  MoveC 1320 to (-42.67, 74.82, -2) mm, rotated rx -180 ry 0 rz 90 deg; joints [75.909, -18.847, 88.976, 0, 19.871, 75.909] to (-41.21, 68.7, -2) mm, rotated rx 180 ry 0 rz 90 deg; joints [75.715, -18.799, 88.77, 0, 20.03, 75.715]
  MoveC 1321 to (-38.99, 66.53, -2) mm, rotated rx 180 ry 0 rz 90 deg; joints [75.66, -18.755, 88.58, 0, 20.175, 75.66] to (-36.48, 64.7, -2) mm, rotated rx -180 ry 0 rz 90 deg; joints [75.62, -18.708, 88.376, 0, 20.331, 75.62]
  MoveL 1322 to (-33.64, 62.89, -2) mm, rotated rx 180 ry 0 rz 90 deg; joints [75.584, -18.654, 88.149, 0, 20.505, 75.584]
  MoveL 1323 to (-13.82, 50.34, -2) mm, rotated rx 180 ry 0 rz 90 deg; joints [75.337, -18.266, 86.548, 0, 21.718, 75.337]
  MoveC 1324 to (-10.3, 48.84, -2) mm, rotated rx -180 ry 0 rz 90 deg; joints [75.318, -18.198, 86.274, 0, 21.924, 75.318] to (-6.48, 48.53, -2) mm, rotated rx 180 ry 0 rz 90 deg; joints [75.34, -18.13, 86.001, 0, 22.129, 75.34]
  MoveL 1325 to (-4.26, 48.7, -2) mm, rotated rx 180 ry 0 rz 90 deg; joints [75.365, -18.091, 85.848, 0, 22.243, 75.365]
  MoveL 1326 to (63.97, 53.62, -2) mm, rotated rx 180 ry 0 rz 90 deg; joints [76.086, -16.793, 80.996, 0, 25.797, 76.086]
  MoveL 1327 to (72, 54.15, -2) mm, rotated rx 180 ry 0 rz 90 deg; joints [76.165, -16.625, 80.404, 0, 26.221, 76.165]
  MoveC 1328 to (76.53, 56.29, -2) mm, rotated rx -180 ry 0 rz 90 deg; joints [76.268, -16.539, 80.104, 0, 26.436, 76.268] to (78.36, 60.94, -2) mm, rotated rx 180 ry 0 rz 90 deg; joints [76.429, -16.524, 80.051, 0, 26.474, 76.429]
  MoveL 1329 to (78.35, 72.49, -2) mm, rotated rx 180 ry 0 rz 90 deg; joints [76.795, -16.584, 80.259, 0, 26.325, 76.795]
  MoveC 1330 to (76.34, 77.27, -2) mm, rotated rx 180 ry 0 rz 90 deg; joints [76.931, -16.651, 80.494, 0, 26.157, 76.931] to (71.55, 79.23, -2) mm, rotated rx 180 ry 0 rz 90 deg; joints [76.958, -16.763, 80.888, 0, 25.875, 76.958]
  MoveC 1331 to (45.96, 79.75, -2) mm, rotated rx 180 ry 0 rz 90 deg; joints [76.784, -17.29, 82.792, 0, 24.498, 76.784] to (20.38, 80.16, -2) mm, rotated rx 180 ry 0 rz 90 deg; joints [76.6, -17.785, 84.654, 0, 23.131, 76.6]
  MoveL 1332 to (20.27, 72.61, -2) mm, rotated rx 180 ry 0 rz 90 deg; joints [76.352, -17.754, 84.532, 0, 23.222, 76.352]
  MoveL 1333 to (20.27, 72.61, 1) mm, rotated rx -180 ry 0 rz 90 deg; joints [76.352, -17.907, 84.632, 0, 23.274, 76.352]
  Establecer velocidad (1000.0 mm/s)
  MoveL 1334 to (20.27, 72.61, 10) mm, rotated rx 180 ry 0 rz 90 deg; joints [76.352, -18.366, 84.932, 0, 23.435, 76.352]
  Establecer velocidad (66.7 mm/s)
  MoveL 1335 to (26.89, 71.36, 10) mm, rotated rx -180 ry 0 rz 90 deg; joints [76.364, -18.234, 84.433, 0, 23.801, 76.364]
  MoveL 1336 to (26.89, 71.36, 1) mm, rotated rx -180 ry 0 rz 90 deg; joints [76.364, -17.776, 84.134, 0, 23.642, 76.364]
  MoveL 1337 to (27.1, 72.86, 0.59) mm, rotated rx -180 ry 0 rz 90 deg; joints [76.415, -17.758, 84.132, 0, 23.626, 76.415]
  MoveL 1338 to (26.94, 74.38, 0.19) mm, rotated rx -180 ry 0 rz 90 deg; joints [76.463, -17.747, 84.156, 0, 23.591, 76.463]
  MoveL 1339 to (26.45, 75.81, -0.22) mm, rotated rx 180 ry 0 rz 90 deg; joints [76.506, -17.743, 84.203, 0, 23.54, 76.506]
  MoveL 1340 to (25.65, 77.11, -0.62) mm, rotated rx -180 ry 0 rz 90 deg; joints [76.542, -17.743, 84.269, 0, 23.474, 76.542]
  MoveL 1341 to (24.58, 78.19, -1.03) mm, rotated rx 180 ry 0 rz 90 deg; joints [76.569, -17.747, 84.351, 0, 23.396, 76.569]
  MoveL 1342 to (23.31, 79.01, -1.44) mm, rotated rx -180 ry 0 rz 90 deg; joints [76.586, -17.754, 84.443, 0, 23.311, 76.586]
  MoveL 1343 to (21.88, 79.53, -1.84) mm, rotated rx 180 ry 0 rz 90 deg; joints [76.591, -17.763, 84.541, 0, 23.222, 76.591]
  MoveL 1344 to (20.37, 79.7, -2.25) mm, rotated rx 180 ry 0 rz 90 deg; joints [76.585, -17.771, 84.638, 0, 23.132, 76.585]
  MoveC 1345 to (-4.74, 80, -2.25) mm, rotated rx 180 ry 0 rz 90 deg; joints [76.396, -18.225, 86.427, 0, 21.799, 76.396] to (-29.85, 80.21, -2.25) mm, rotated rx 180 ry 0 rz 90 deg; joints [76.198, -18.65, 88.179, 0, 20.471, 76.198]
  MoveL 1346 to (-30.8, 80.2, -2.25) mm, rotated rx -180 ry 0 rz 90 deg; joints [76.19, -18.665, 88.244, 0, 20.421, 76.19]
  MoveC 1347 to (-34.29, 79.93, -2.25) mm, rotated rx -180 ry 0 rz 90 deg; joints [76.152, -18.721, 88.48, 0, 20.241, 76.152] to (-37.7, 79.16, -2.25) mm, rotated rx -180 ry 0 rz 90 deg; joints [76.097, -18.772, 88.701, 0, 20.072, 76.097]
  MoveC 1348 to (-42.06, 74.54, -2.25) mm, rotated rx -180 ry 0 rz 90 deg; joints [75.904, -18.823, 88.921, 0, 19.903, 75.904] to (-40.34, 68.41, -2.25) mm, rotated rx 180 ry 0 rz 90 deg; joints [75.712, -18.771, 88.697, 0, 20.074, 75.712]
  MoveC 1349 to (-38.41, 66.69, -2.25) mm, rotated rx -180 ry 0 rz 90 deg; joints [75.671, -18.734, 88.535, 0, 20.199, 75.671] to (-36.32, 65.17, -2.25) mm, rotated rx 180 ry 0 rz 90 deg; joints [75.638, -18.694, 88.365, 0, 20.329, 75.638]
  MoveL 1350 to (-33.64, 63.44, -2.25) mm, rotated rx 180 ry 0 rz 90 deg; joints [75.602, -18.643, 88.15, 0, 20.493, 75.602]
  MoveL 1351 to (-13.47, 50.68, -2.25) mm, rotated rx -180 ry 0 rz 90 deg; joints [75.351, -18.249, 86.522, 0, 21.727, 75.351]
  MoveC 1352 to (-10.21, 49.29, -2.25) mm, rotated rx -180 ry 0 rz 90 deg; joints [75.333, -18.186, 86.268, 0, 21.918, 75.333] to (-6.69, 48.98, -2.25) mm, rotated rx 180 ry 0 rz 90 deg; joints [75.354, -18.123, 86.015, 0, 22.108, 75.354]
  MoveL 1353 to (56.07, 53.54, -2.25) mm, rotated rx 180 ry 0 rz 90 deg; joints [76.021, -16.944, 81.572, 0, 25.372, 76.021]
  MoveL 1354 to (72.01, 54.62, -2.25) mm, rotated rx 180 ry 0 rz 90 deg; joints [76.18, -16.615, 80.404, 0, 26.211, 76.18]
  MoveC 1355 to (76.2, 56.62, -2.25) mm, rotated rx -180 ry 0 rz 90 deg; joints [76.276, -16.536, 80.126, 0, 26.41, 76.276] to (77.91, 60.93, -2.25) mm, rotated rx -180 ry 0 rz 90 deg; joints [76.426, -16.521, 80.076, 0, 26.445, 76.426]
  MoveL 1356 to (77.91, 71.55, -2.25) mm, rotated rx -180 ry 0 rz 90 deg; joints [76.762, -16.576, 80.267, 0, 26.309, 76.762]
  MoveL 1357 to (77.9, 72.49, -2.25) mm, rotated rx 180 ry 0 rz 90 deg; joints [76.792, -16.581, 80.284, 0, 26.297, 76.792]
  MoveC 1358 to (76.02, 76.94, -2.25) mm, rotated rx 180 ry 0 rz 90 deg; joints [76.919, -16.644, 80.504, 0, 26.139, 76.919] to (71.55, 78.78, -2.25) mm, rotated rx -180 ry 0 rz 90 deg; joints [76.944, -16.748, 80.872, 0, 25.876, 76.944]
  MoveC 1359 to (45.96, 79.28, -2.25) mm, rotated rx 180 ry 0 rz 90 deg; joints [76.769, -17.276, 82.776, 0, 24.499, 76.769] to (20.37, 79.7, -2.25) mm, rotated rx 180 ry 0 rz 90 deg; joints [76.585, -17.771, 84.638, 0, 23.132, 76.585]
  MoveL 1360 to (20.26, 72.14, -2.25) mm, rotated rx 180 ry 0 rz 90 deg; joints [76.337, -17.739, 84.516, 0, 23.223, 76.337]
  MoveL 1361 to (20.26, 72.14, 0.75) mm, rotated rx 180 ry 0 rz 90 deg; joints [76.337, -17.892, 84.616, 0, 23.276, 76.337]
  Establecer velocidad (1000.0 mm/s)
  MoveL 1362 to (20.26, 72.14, 10) mm, rotated rx -180 ry 0 rz 90 deg; joints [76.337, -18.364, 84.924, 0, 23.441, 76.337]
  Establecer velocidad (66.7 mm/s)
  MoveL 1363 to (37.42, 27.37, 10) mm, rotated rx -180 ry 0 rz 90 deg; joints [75.031, -17.807, 82.856, 0, 24.951, 75.031]
  MoveL 1364 to (37.42, 27.37, 1) mm, rotated rx 180 ry 0 rz 90 deg; joints [75.031, -17.351, 82.556, 0, 24.795, 75.031]
  MoveL 1365 to (37.57, 28.88, 0.59) mm, rotated rx 180 ry 0 rz 90 deg; joints [75.08, -17.335, 82.561, 0, 24.774, 75.08]
  MoveL 1366 to (37.34, 30.39, 0.19) mm, rotated rx 180 ry 0 rz 90 deg; joints [75.127, -17.327, 82.593, 0, 24.734, 75.127]
  MoveL 1367 to (36.79, 31.8, -0.22) mm, rotated rx -180 ry 0 rz 90 deg; joints [75.167, -17.325, 82.647, 0, 24.678, 75.167]
  MoveL 1368 to (35.94, 33.06, -0.62) mm, rotated rx 180 ry 0 rz 90 deg; joints [75.2, -17.328, 82.72, 0, 24.608, 75.2]
  MoveL 1369 to (34.84, 34.1, -1.03) mm, rotated rx 180 ry 0 rz 90 deg; joints [75.224, -17.335, 82.807, 0, 24.528, 75.224]
  MoveL 1370 to (33.53, 34.87, -1.44) mm, rotated rx 180 ry 0 rz 90 deg; joints [75.238, -17.344, 82.903, 0, 24.441, 75.238]
  MoveL 1371 to (32.08, 35.33, -1.84) mm, rotated rx -180 ry 0 rz 90 deg; joints [75.241, -17.354, 83.003, 0, 24.351, 75.241]
  MoveL 1372 to (30.56, 35.43, -2.25) mm, rotated rx -180 ry 0 rz 90 deg; joints [75.231, -17.364, 83.101, 0, 24.262, 75.231]
  MoveL 1373 to (8.05, 34.82, -2.25) mm, rotated rx 180 ry 0 rz 90 deg; joints [75.018, -17.789, 84.707, 0, 23.081, 75.018]
  MoveL 1374 to (7.11, 34.77, -2.25) mm, rotated rx -180 ry 0 rz 90 deg; joints [75.008, -17.806, 84.774, 0, 23.032, 75.008]
  MoveC 1375 to (3.74, 33.88, -2.25) mm, rotated rx 180 ry 0 rz 90 deg; joints [74.949, -17.863, 84.996, 0, 22.868, 74.949] to (1, 31.75, -2.25) mm, rotated rx 180 ry 0 rz 90 deg; joints [74.856, -17.903, 85.149, 0, 22.753, 74.856]
  MoveC 1376 to (-0.42, 28.07, -2.25) mm, rotated rx 180 ry 0 rz 90 deg; joints [74.723, -17.91, 85.179, 0, 22.731, 74.723] to (0.08, 24.17, -2.25) mm, rotated rx -180 ry 0 rz 90 deg; joints [74.6, -17.882, 85.068, 0, 22.814, 74.6]
  MoveL 1377 to (6.28, 7.11, -2.25) mm, rotated rx 180 ry 0 rz 90 deg; joints [74.103, -17.679, 84.288, 0, 23.391, 74.103]
  MoveC 1378 to (7.37, 5.07, -2.25) mm, rotated rx 180 ry 0 rz 90 deg; joints [74.047, -17.648, 84.169, 0, 23.479, 74.047] to (9, 3.43, -2.25) mm, rotated rx -180 ry 0 rz 90 deg; joints [74.01, -17.609, 84.02, 0, 23.589, 74.01]
  MoveL 1379 to (26.06, -9.85, -2.25) mm, rotated rx -180 ry 0 rz 90 deg; joints [73.742, -17.205, 82.517, 0, 24.688, 73.742]
  MoveL 1380 to (26.62, -10.26, -2.25) mm, rotated rx -180 ry 0 rz 90 deg; joints [73.735, -17.191, 82.467, 0, 24.724, 73.735]
  MoveC 1381 to (31.94, -11.66, -2.25) mm, rotated rx -180 ry 0 rz 90 deg; joints [73.74, -17.077, 82.051, 0, 25.026, 73.74] to (36.8, -9.09, -2.25) mm, rotated rx 180 ry 0 rz 90 deg; joints [73.866, -16.994, 81.751, 0, 25.243, 73.866]
  MoveL 1382 to (37.43, -8.35, -2.25) mm, rotated rx 180 ry 0 rz 90 deg; joints [73.895, -16.986, 81.72, 0, 25.265, 73.895]
  MoveL 1383 to (60.11, 23.22, -2.25) mm, rotated rx 180 ry 0 rz 90 deg; joints [75.091, -16.697, 80.693, 0, 26.004, 75.091]
  MoveC 1384 to (61.33, 25.15, -2.25) mm, rotated rx 180 ry 0 rz 90 deg; joints [75.162, -16.682, 80.64, 0, 26.042, 75.162] to (62.23, 27.25, -2.25) mm, rotated rx 180 ry 0 rz 90 deg; joints [75.236, -16.675, 80.614, 0, 26.061, 75.236]
  MoveC 1385 to (61.82, 32.4, -2.25) mm, rotated rx 180 ry 0 rz 90 deg; joints [75.396, -16.712, 80.745, 0, 25.967, 75.396] to (57.77, 35.62, -2.25) mm, rotated rx 180 ry 0 rz 90 deg; joints [75.464, -16.815, 81.109, 0, 25.706, 75.464]
  MoveC 1386 to (55.91, 35.98, -2.25) mm, rotated rx 180 ry 0 rz 90 deg; joints [75.46, -16.855, 81.254, 0, 25.602, 75.46] to (54.02, 36.06, -2.25) mm, rotated rx -180 ry 0 rz 90 deg; joints [75.447, -16.895, 81.395, 0, 25.5, 75.447]
  MoveL 1387 to (30.56, 35.43, -2.25) mm, rotated rx -180 ry 0 rz 90 deg; joints [75.231, -17.364, 83.101, 0, 24.262, 75.231]
  MoveL 1388 to (30.77, 27.88, -2.25) mm, rotated rx -180 ry 0 rz 90 deg; joints [74.99, -17.32, 82.941, 0, 24.379, 74.99]
  MoveL 1389 to (30.77, 27.88, 0.75) mm, rotated rx 180 ry 0 rz 90 deg; joints [74.99, -17.473, 83.042, 0, 24.431, 74.99]
  Establecer velocidad (1000.0 mm/s)
  MoveL 1390 to (30.77, 27.88, 10) mm, rotated rx 180 ry 0 rz 90 deg; joints [74.99, -17.942, 83.35, 0, 24.592, 74.99]
  Establecer velocidad (66.7 mm/s)
  MoveL 1391 to (70.1, -30.05, 10) mm, rotated rx -180 ry 0 rz 90 deg; joints [73.515, -16.77, 79.233, 0, 27.537, 73.515]
  MoveL 1392 to (70.1, -30.05, 1) mm, rotated rx 180 ry 0 rz 90 deg; joints [73.515, -16.32, 78.931, 0, 27.389, 73.515]
  MoveL 1393 to (71.61, -30.24, 0.59) mm, rotated rx -180 ry 0 rz 90 deg; joints [73.523, -16.265, 78.799, 0, 27.465, 73.523]
  MoveL 1394 to (73.12, -30.06, 0.19) mm, rotated rx 180 ry 0 rz 90 deg; joints [73.542, -16.212, 78.676, 0, 27.536, 73.542]
  MoveL 1395 to (74.55, -29.55, -0.22) mm, rotated rx 180 ry 0 rz 90 deg; joints [73.571, -16.163, 78.565, 0, 27.598, 73.571]
  MoveL 1396 to (75.83, -28.73, -0.62) mm, rotated rx -180 ry 0 rz 90 deg; joints [73.608, -16.119, 78.472, 0, 27.647, 73.608]
  MoveL 1397 to (76.9, -27.65, -1.03) mm, rotated rx -180 ry 0 rz 90 deg; joints [73.651, -16.082, 78.401, 0, 27.681, 73.651]
  MoveL 1398 to (77.7, -26.36, -1.44) mm, rotated rx 180 ry 0 rz 90 deg; joints [73.698, -16.052, 78.355, 0, 27.697, 73.698]
  MoveL 1399 to (78.2, -24.93, -1.84) mm, rotated rx 180 ry 0 rz 90 deg; joints [73.746, -16.03, 78.335, 0, 27.695, 73.746]
  MoveL 1400 to (78.34, -23.41, -2.25) mm, rotated rx 180 ry 0 rz 90 deg; joints [73.794, -16.016, 78.344, 0, 27.672, 73.794]
  MoveL 1401 to (78.34, -5.21, -2.25) mm, rotated rx -180 ry 0 rz 90 deg; joints [74.357, -16.133, 78.739, 0, 27.394, 74.357]
  MoveC 1402 to (78.23, -2.56, -2.25) mm, rotated rx -180 ry 0 rz 90 deg; joints [74.439, -16.152, 78.804, 0, 27.348, 74.439] to (77.84, 0.06, -2.25) mm, rotated rx -180 ry 0 rz 90 deg; joints [74.517, -16.177, 78.888, 0, 27.288, 74.517]
  MoveC 1403 to (74.21, 4.2, -2.25) mm, rotated rx 180 ry 0 rz 90 deg; joints [74.614, -16.282, 79.249, 0, 27.033, 74.614] to (68.7, 4.38, -2.25) mm, rotated rx -180 ry 0 rz 90 deg; joints [74.572, -16.404, 79.668, 0, 26.736, 74.572]
  MoveC 1404 to (66.87, 2.88, -2.25) mm, rotated rx 180 ry 0 rz 90 deg; joints [74.51, -16.434, 79.774, 0, 26.66, 74.51] to (65.31, 1.09, -2.25) mm, rotated rx 180 ry 0 rz 90 deg; joints [74.44, -16.458, 79.854, 0, 26.603, 74.44]
  MoveL 1405 to (64.15, -0.47, -2.25) mm, rotated rx 180 ry 0 rz 90 deg; joints [74.381, -16.473, 79.908, 0, 26.565, 74.381]
  MoveL 1406 to (48.95, -21.32, -2.25) mm, rotated rx 180 ry 0 rz 90 deg; joints [73.592, -16.669, 80.594, 0, 26.075, 73.592]
  MoveL 1407 to (48.51, -21.97, -2.25) mm, rotated rx 180 ry 0 rz 90 deg; joints [73.568, -16.674, 80.613, 0, 26.062, 73.568]
  MoveC 1408 to (47.28, -26.49, -2.25) mm, rotated rx -180 ry 0 rz 90 deg; joints [73.415, -16.672, 80.605, 0, 26.068, 73.415] to (49.04, -30.82, -2.25) mm, rotated rx 180 ry 0 rz 90 deg; joints [73.296, -16.608, 80.378, 0, 26.23, 73.296]
  MoveL 1409 to (49.75, -31.64, -2.25) mm, rotated rx -180 ry 0 rz 90 deg; joints [73.277, -16.588, 80.308, 0, 26.28, 73.277]
  MoveL 1410 to (64.94, -48.8, -2.25) mm, rotated rx 180 ry 0 rz 90 deg; joints [72.888, -16.146, 78.784, 0, 27.362, 72.888]
  MoveL 1411 to (66.07, -50.02, -2.25) mm, rotated rx -180 ry 0 rz 90 deg; joints [72.861, -16.112, 78.67, 0, 27.443, 72.861]
  MoveC 1412 to (67.73, -51.48, -2.25) mm, rotated rx 180 ry 0 rz 90 deg; joints [72.832, -16.066, 78.511, 0, 27.555, 72.832] to (69.65, -52.58, -2.25) mm, rotated rx -180 ry 0 rz 90 deg; joints [72.817, -16.015, 78.34, 0, 27.675, 72.817]
  MoveC 1413 to (75.13, -51.63, -2.25) mm, rotated rx 180 ry 0 rz 90 deg; joints [72.898, -15.898, 77.947, 0, 27.951, 72.898] to (78.06, -46.91, -2.25) mm, rotated rx 180 ry 0 rz 90 deg; joints [73.07, -15.865, 77.834, 0, 28.031, 73.07]
  MoveC 1414 to (78.27, -45.02, -2.25) mm, rotated rx 180 ry 0 rz 90 deg; joints [73.13, -15.873, 77.862, 0, 28.011, 73.13] to (78.34, -43.12, -2.25) mm, rotated rx 180 ry 0 rz 90 deg; joints [73.188, -15.884, 77.9, 0, 27.984, 73.188]
  MoveL 1415 to (78.34, -23.41, -2.25) mm, rotated rx 180 ry 0 rz 90 deg; joints [73.794, -16.016, 78.344, 0, 27.672, 73.794]
  MoveL 1416 to (70.79, -23.41, -2.25) mm, rotated rx -180 ry 0 rz 90 deg; joints [73.726, -16.185, 78.916, 0, 27.269, 73.726]
  MoveL 1417 to (70.79, -23.41, 0.75) mm, rotated rx 180 ry 0 rz 90 deg; joints [73.726, -16.335, 79.018, 0, 27.317, 73.726]
  Establecer velocidad (1000.0 mm/s)
  MoveL 1418 to (70.79, -23.41, 10) mm, rotated rx 180 ry 0 rz 90 deg; joints [73.726, -16.798, 79.328, 0, 27.47, 73.726]
  Establecer velocidad (66.7 mm/s)
  MoveL 1419 to (18.87, -71.64, 10) mm, rotated rx -180 ry 0 rz 90 deg; joints [71.724, -17.584, 82.056, 0, 25.528, 71.724]
  MoveL 1420 to (18.87, -71.64, 1) mm, rotated rx 180 ry 0 rz 90 deg; joints [71.724, -17.129, 81.756, 0, 25.374, 71.724]
  MoveL 1421 to (18.7, -73.15, 0.59) mm, rotated rx -180 ry 0 rz 90 deg; joints [71.675, -17.102, 81.718, 0, 25.384, 71.675]
  MoveL 1422 to (18.9, -74.65, 0.19) mm, rotated rx 180 ry 0 rz 90 deg; joints [71.63, -17.068, 81.654, 0, 25.413, 71.63]
  MoveL 1423 to (19.42, -76.08, -0.22) mm, rotated rx -180 ry 0 rz 90 deg; joints [71.591, -17.027, 81.568, 0, 25.459, 71.591]
  MoveL 1424 to (20.25, -77.35, -0.62) mm, rotated rx 180 ry 0 rz 90 deg; joints [71.56, -16.981, 81.464, 0, 25.517, 71.56]
  MoveL 1425 to (21.34, -78.41, -1.03) mm, rotated rx 180 ry 0 rz 90 deg; joints [71.538, -16.931, 81.345, 0, 25.586, 71.538]
  MoveL 1426 to (22.63, -79.2, -1.44) mm, rotated rx 180 ry 0 rz 90 deg; joints [71.527, -16.879, 81.218, 0, 25.66, 71.527]
  MoveL 1427 to (24.07, -79.69, -1.84) mm, rotated rx -180 ry 0 rz 90 deg; joints [71.527, -16.825, 81.088, 0, 25.737, 71.527]
  MoveL 1428 to (25.59, -79.81, -2.25) mm, rotated rx -180 ry 0 rz 90 deg; joints [71.539, -16.773, 80.961, 0, 25.812, 71.539]
  MoveL 1429 to (46.91, -79.61, -2.25) mm, rotated rx -180 ry 0 rz 90 deg; joints [71.764, -16.325, 79.398, 0, 26.928, 71.764]
  MoveL 1430 to (53.54, -79.52, -2.25) mm, rotated rx 180 ry 0 rz 90 deg; joints [71.833, -16.182, 78.906, 0, 27.276, 71.833]
  MoveC 1431 to (56.29, -79.18, -2.25) mm, rotated rx -180 ry 0 rz 90 deg; joints [71.871, -16.124, 78.709, 0, 27.415, 71.871] to (58.87, -78.18, -2.25) mm, rotated rx 180 ry 0 rz 90 deg; joints [71.928, -16.074, 78.54, 0, 27.534, 71.928]
  MoveC 1432 to (61.62, -73.98, -2.25) mm, rotated rx -180 ry 0 rz 90 deg; joints [72.083, -16.043, 78.435, 0, 27.608, 72.083] to (60.79, -69.03, -2.25) mm, rotated rx -180 ry 0 rz 90 deg; joints [72.227, -16.097, 78.618, 0, 27.479, 72.227]
  MoveC 1433 to (59.74, -67.45, -2.25) mm, rotated rx 180 ry 0 rz 90 deg; joints [72.265, -16.132, 78.735, 0, 27.397, 72.265] to (58.56, -65.96, -2.25) mm, rotated rx -180 ry 0 rz 90 deg; joints [72.299, -16.168, 78.859, 0, 27.309, 72.299]
  MoveL 1434 to (29.78, -32.69, -2.25) mm, rotated rx 180 ry 0 rz 90 deg; joints [73.055, -16.994, 81.751, 0, 25.243, 73.055]
  MoveL 1435 to (28.9, -31.85, -2.25) mm, rotated rx 180 ry 0 rz 90 deg; joints [73.073, -17.017, 81.834, 0, 25.183, 73.073]
  MoveL 1436 to (24.17, -28.06, -2.25) mm, rotated rx 180 ry 0 rz 90 deg; joints [73.147, -17.135, 82.262, 0, 24.873, 73.147]
  MoveL 1437 to (14.55, -20.37, -2.25) mm, rotated rx -180 ry 0 rz 90 deg; joints [73.299, -17.369, 83.123, 0, 24.247, 73.299]
  MoveL 1438 to (13.74, -19.78, -2.25) mm, rotated rx -180 ry 0 rz 90 deg; joints [73.31, -17.388, 83.193, 0, 24.195, 73.31]
  MoveC 1439 to (10.6, -18.25, -2.25) mm, rotated rx -180 ry 0 rz 90 deg; joints [73.329, -17.458, 83.452, 0, 24.006, 73.329] to (7.11, -18.01, -2.25) mm, rotated rx 180 ry 0 rz 90 deg; joints [73.303, -17.525, 83.706, 0, 23.819, 73.303]
  MoveC 1440 to (3.54, -19.84, -2.25) mm, rotated rx 180 ry 0 rz 90 deg; joints [73.21, -17.582, 83.921, 0, 23.662, 73.21] to (1.39, -23.22, -2.25) mm, rotated rx 180 ry 0 rz 90 deg; joints [73.081, -17.604, 84.001, 0, 23.602, 73.081]
  MoveL 1441 to (1.06, -24.17, -2.25) mm, rotated rx 180 ry 0 rz 90 deg; joints [73.047, -17.604, 84.004, 0, 23.601, 73.047]
  MoveL 1442 to (-4.47, -45.01, -2.25) mm, rotated rx 180 ry 0 rz 90 deg; joints [72.326, -17.586, 83.935, 0, 23.651, 72.326]
  MoveL 1443 to (-11.01, -69.65, -2.25) mm, rotated rx -180 ry 0 rz 90 deg; joints [71.474, -17.558, 83.828, 0, 23.73, 71.474]
  MoveL 1444 to (-11.23, -70.6, -2.25) mm, rotated rx -180 ry 0 rz 90 deg; joints [71.441, -17.556, 83.821, 0, 23.735, 71.441]
  MoveC 1445 to (-10.15, -76.46, -2.25) mm, rotated rx 180 ry 0 rz 90 deg; joints [71.267, -17.499, 83.605, 0, 23.893, 71.267] to (-5.21, -79.8, -2.25) mm, rotated rx 180 ry 0 rz 90 deg; joints [71.214, -17.384, 83.176, 0, 24.208, 71.214]
  MoveC 1446 to (-3.8, -80.03, -2.25) mm, rotated rx -180 ry 0 rz 90 deg; joints [71.223, -17.355, 83.07, 0, 24.285, 71.223] to (-2.37, -80.08, -2.25) mm, rotated rx -180 ry 0 rz 90 deg; joints [71.236, -17.327, 82.967, 0, 24.36, 71.236]
  MoveL 1447 to (25.59, -79.81, -2.25) mm, rotated rx -180 ry 0 rz 90 deg; joints [71.539, -16.773, 80.961, 0, 25.812, 71.539]
  MoveL 1448 to (25.51, -72.27, -2.25) mm, rotated rx 180 ry 0 rz 90 deg; joints [71.773, -16.826, 81.149, 0, 25.677, 71.773]
  MoveL 1449 to (25.51, -72.27, 0.75) mm, rotated rx -180 ry 0 rz 90 deg; joints [71.773, -16.977, 81.25, 0, 25.727, 71.773]
  Establecer velocidad (1000.0 mm/s)
  MoveL 1450 to (25.51, -72.27, 10) mm, rotated rx -180 ry 0 rz 90 deg; joints [71.773, -17.444, 81.559, 0, 25.885, 71.773]
  Establecer velocidad (66.7 mm/s)
  MoveL 1451 to (-60.11, -71.82, 10) mm, rotated rx 180 ry 0 rz 90 deg; joints [70.867, -19.042, 87.581, 0, 21.461, 70.867]
  MoveL 1452 to (-60.11, -71.82, 1) mm, rotated rx 180 ry 0 rz 90 deg; joints [70.867, -18.577, 87.282, 0, 21.295, 70.867]
  MoveL 1453 to (-60.28, -73.32, 0.59) mm, rotated rx 180 ry 0 rz 90 deg; joints [70.816, -18.55, 87.245, 0, 21.305, 70.816]
  MoveL 1454 to (-60.09, -74.83, 0.19) mm, rotated rx 180 ry 0 rz 90 deg; joints [70.769, -18.517, 87.182, 0, 21.335, 70.769]
  MoveL 1455 to (-59.57, -76.26, -0.22) mm, rotated rx 180 ry 0 rz 90 deg; joints [70.729, -18.479, 87.099, 0, 21.38, 70.729]
  MoveL 1456 to (-58.74, -77.54, -0.62) mm, rotated rx 180 ry 0 rz 90 deg; joints [70.697, -18.437, 87, 0, 21.438, 70.697]
  MoveL 1457 to (-57.65, -78.6, -1.03) mm, rotated rx -180 ry 0 rz 90 deg; joints [70.675, -18.392, 86.887, 0, 21.505, 70.675]
  MoveL 1458 to (-56.36, -79.39, -1.44) mm, rotated rx 180 ry 0 rz 90 deg; joints [70.664, -18.345, 86.766, 0, 21.579, 70.664]
  MoveL 1459 to (-54.92, -79.88, -1.84) mm, rotated rx 180 ry 0 rz 90 deg; joints [70.664, -18.297, 86.643, 0, 21.654, 70.664]
  MoveL 1460 to (-53.41, -80.01, -2.25) mm, rotated rx 180 ry 0 rz 90 deg; joints [70.677, -18.249, 86.523, 0, 21.726, 70.677]
  MoveL 1461 to (-35.27, -79.87, -2.25) mm, rotated rx -180 ry 0 rz 90 deg; joints [70.885, -17.936, 85.28, 0, 22.656, 70.885]
  MoveC 1462 to (-29.73, -77.98, -2.25) mm, rotated rx -180 ry 0 rz 90 deg; joints [71.006, -17.849, 84.941, 0, 22.908, 71.006] to (-26.4, -73.16, -2.25) mm, rotated rx -180 ry 0 rz 90 deg; joints [71.196, -17.819, 84.824, 0, 22.994, 71.196]
  MoveL 1463 to (-26.21, -72.49, -2.25) mm, rotated rx 180 ry 0 rz 90 deg; joints [71.22, -17.82, 84.827, 0, 22.993, 71.22]
  MoveL 1464 to (-13.74, -24.57, -2.25) mm, rotated rx -180 ry 0 rz 90 deg; joints [72.889, -17.875, 85.041, 0, 22.834, 72.889]
  MoveL 1465 to (-13.64, -24.17, -2.25) mm, rotated rx 180 ry 0 rz 90 deg; joints [72.903, -17.875, 85.042, 0, 22.833, 72.903]
  MoveC 1466 to (-13.44, -19.72, -2.25) mm, rotated rx 180 ry 0 rz 90 deg; joints [73.048, -17.896, 85.123, 0, 22.773, 73.048] to (-15.2, -15.64, -2.25) mm, rotated rx 180 ry 0 rz 90 deg; joints [73.163, -17.95, 85.334, 0, 22.616, 73.163]
  MoveC 1467 to (-19.03, -13.05, -2.25) mm, rotated rx 180 ry 0 rz 90 deg; joints [73.21, -18.032, 85.657, 0, 22.375, 73.21] to (-23.65, -12.75, -2.25) mm, rotated rx -180 ry 0 rz 90 deg; joints [73.174, -18.115, 85.985, 0, 22.13, 73.174]
  MoveL 1468 to (-26.06, -13.23, -2.25) mm, rotated rx 180 ry 0 rz 90 deg; joints [73.134, -18.155, 86.142, 0, 22.012, 73.134]
  MoveL 1469 to (-73.46, -23.33, -2.25) mm, rotated rx 180 ry 0 rz 90 deg; joints [72.316, -18.878, 89.16, 0, 19.718, 72.316]
  MoveC 1470 to (-78.73, -26.56, -2.25) mm, rotated rx 180 ry 0 rz 90 deg; joints [72.152, -18.943, 89.443, 0, 19.5, 72.152] to (-80.79, -32.38, -2.25) mm, rotated rx 180 ry 0 rz 90 deg; joints [71.935, -18.945, 89.455, 0, 19.491, 71.935]
  MoveL 1471 to (-80.79, -70.98, -2.25) mm, rotated rx -180 ry 0 rz 90 deg; joints [70.658, -18.745, 88.583, 0, 20.162, 70.658]
  MoveC 1472 to (-78.08, -77.49, -2.25) mm, rotated rx -180 ry 0 rz 90 deg; joints [70.476, -18.667, 88.249, 0, 20.418, 70.476] to (-71.54, -80.15, -2.25) mm, rotated rx 180 ry 0 rz 90 deg; joints [70.465, -18.548, 87.748, 0, 20.8, 70.465]
  MoveL 1473 to (-53.41, -80.01, -2.25) mm, rotated rx 180 ry 0 rz 90 deg; joints [70.677, -18.249, 86.523, 0, 21.726, 70.677]
  MoveL 1474 to (-53.47, -72.46, -2.25) mm, rotated rx 180 ry 0 rz 90 deg; joints [70.92, -18.295, 86.706, 0, 21.588, 70.92]
  MoveL 1475 to (-53.47, -72.46, 0.75) mm, rotated rx 180 ry 0 rz 90 deg; joints [70.92, -18.449, 86.807, 0, 21.642, 70.92]
  Establecer velocidad (1000.0 mm/s)
  MoveL 1476 to (-53.47, -72.46, 10) mm, rotated rx 180 ry 0 rz 90 deg; joints [70.92, -18.926, 87.114, 0, 21.812, 70.92]
  Establecer velocidad (66.7 mm/s)
  MoveL 1477 to (-72.55, 36.29, 10) mm, rotated rx 180 ry 0 rz 90 deg; joints [74.332, -19.775, 90.703, 0, 19.073, 74.332]
  MoveL 1478 to (-72.55, 36.29, 1) mm, rotated rx 180 ry 0 rz 90 deg; joints [74.332, -19.304, 90.403, 0, 18.9, 74.332]
  MoveL 1479 to (-74.05, 36.47, 0.59) mm, rotated rx -180 ry 0 rz 90 deg; joints [74.324, -19.305, 90.494, 0, 18.811, 74.324]
  MoveL 1480 to (-75.56, 36.29, 0.19) mm, rotated rx 180 ry 0 rz 90 deg; joints [74.303, -19.305, 90.578, 0, 18.728, 74.303]
  MoveL 1481 to (-76.99, 35.78, -0.22) mm, rotated rx 180 ry 0 rz 90 deg; joints [74.272, -19.303, 90.65, 0, 18.653, 74.272]
  MoveL 1482 to (-78.28, 34.96, -0.62) mm, rotated rx -180 ry 0 rz 90 deg; joints [74.232, -19.297, 90.706, 0, 18.59, 74.232]
  MoveL 1483 to (-79.34, 33.88, -1.03) mm, rotated rx 180 ry 0 rz 90 deg; joints [74.185, -19.286, 90.743, 0, 18.543, 74.185]
  MoveL 1484 to (-80.15, 32.59, -1.44) mm, rotated rx -180 ry 0 rz 90 deg; joints [74.133, -19.271, 90.759, 0, 18.512, 74.133]
  MoveL 1485 to (-80.65, 31.16, -1.84) mm, rotated rx -180 ry 0 rz 90 deg; joints [74.079, -19.251, 90.751, 0, 18.5, 74.079]
  MoveL 1486 to (-80.79, 29.64, -2.25) mm, rotated rx -180 ry 0 rz 90 deg; joints [74.026, -19.226, 90.718, 0, 18.508, 74.026]
  MoveL 1487 to (-80.78, 0.47, -2.25) mm, rotated rx -180 ry 0 rz 90 deg; joints [73.037, -19.1, 90.144, 0, 18.955, 73.037]
  MoveC 1488 to (-77.75, -6.36, -2.25) mm, rotated rx -180 ry 0 rz 90 deg; joints [72.838, -19.024, 89.803, 0, 19.221, 72.838] to (-70.6, -8.55, -2.25) mm, rotated rx -180 ry 0 rz 90 deg; joints [72.839, -18.905, 89.279, 0, 19.626, 72.839]
  MoveL 1489 to (-69.65, -8.43, -2.25) mm, rotated rx -180 ry 0 rz 90 deg; joints [72.853, -18.892, 89.218, 0, 19.673, 72.853]
  MoveL 1490 to (-63.02, -6.92, -2.25) mm, rotated rx 180 ry 0 rz 90 deg; joints [72.971, -18.796, 88.803, 0, 19.993, 72.971]
  MoveL 1491 to (-19.43, 3.11, -2.25) mm, rotated rx 180 ry 0 rz 90 deg; joints [73.733, -18.124, 86.019, 0, 22.105, 73.733]
  MoveC 1492 to (-13.57, 7.44, -2.25) mm, rotated rx 180 ry 0 rz 90 deg; joints [73.929, -18.042, 85.697, 0, 22.345, 73.929] to (-12.82, 14.69, -2.25) mm, rotated rx 180 ry 0 rz 90 deg; joints [74.173, -18.066, 85.79, 0, 22.276, 74.173]
  MoveL 1493 to (-13.12, 15.64, -2.25) mm, rotated rx 180 ry 0 rz 90 deg; joints [74.201, -18.076, 85.83, 0, 22.246, 74.201]
  MoveL 1494 to (-19.79, 34.25, -2.25) mm, rotated rx 180 ry 0 rz 90 deg; joints [74.752, -18.282, 86.657, 0, 21.626, 74.752]
  MoveC 1495 to (-21.29, 36.95, -2.25) mm, rotated rx 180 ry 0 rz 90 deg; joints [74.828, -18.321, 86.812, 0, 21.509, 74.828] to (-23.58, 39.01, -2.25) mm, rotated rx -180 ry 0 rz 90 deg; joints [74.876, -18.369, 87.01, 0, 21.359, 74.876]
  MoveL 1496 to (-65.41, 65.86, -2.25) mm, rotated rx -180 ry 0 rz 90 deg; joints [75.406, -19.146, 90.352, 0, 18.794, 75.406]
  MoveL 1497 to (-66.15, 66.33, -2.25) mm, rotated rx -180 ry 0 rz 90 deg; joints [75.416, -19.158, 90.41, 0, 18.749, 75.416]
  MoveC 1498 to (-69.29, 67.73, -2.25) mm, rotated rx 180 ry 0 rz 90 deg; joints [75.436, -19.21, 90.645, 0, 18.565, 75.436] to (-72.7, 68.19, -2.25) mm, rotated rx 180 ry 0 rz 90 deg; joints [75.421, -19.261, 90.881, 0, 18.38, 75.421]
  MoveC 1499 to (-76.86, 66.93, -2.25) mm, rotated rx -180 ry 0 rz 90 deg; joints [75.34, -19.316, 91.136, 0, 18.179, 75.34] to (-79.72, 63.66, -2.25) mm, rotated rx -180 ry 0 rz 90 deg; joints [75.202, -19.344, 91.269, 0, 18.075, 75.202]
  MoveC 1500 to (-80.52, 61.3, -2.25) mm, rotated rx -180 ry 0 rz 90 deg; joints [75.113, -19.347, 91.281, 0, 18.066, 75.113] to (-80.79, 58.82, -2.25) mm, rotated rx 180 ry 0 rz 90 deg; joints [75.025, -19.341, 91.255, 0, 18.086, 75.025]
  MoveL 1501 to (-80.79, 29.64, -2.25) mm, rotated rx -180 ry 0 rz 90 deg; joints [74.026, -19.226, 90.718, 0, 18.508, 74.026]
  MoveL 1502 to (-73.24, 29.65, -2.25) mm, rotated rx -180 ry 0 rz 90 deg; joints [74.1, -19.116, 90.215, 0, 18.901, 74.1]
  MoveL 1503 to (-73.24, 29.65, 0.75) mm, rotated rx -180 ry 0 rz 90 deg; joints [74.1, -19.273, 90.316, 0, 18.957, 74.1]
  Establecer velocidad (1000.0 mm/s)
  MoveL 1504 to (-73.24, 29.65, 10) mm, rotated rx 180 ry 0 rz 90 deg; joints [74.1, -19.758, 90.623, 0, 19.134, 74.1]
  Establecer velocidad (66.7 mm/s)
  MoveL 1505 to (-72.12, 36.29, 10) mm, rotated rx -180 ry 0 rz 90 deg; joints [74.336, -19.769, 90.674, 0, 19.095, 74.336]
  MoveL 1506 to (-72.12, 36.29, 0.75) mm, rotated rx -180 ry 0 rz 90 deg; joints [74.336, -19.284, 90.366, 0, 18.918, 74.336]
  MoveL 1507 to (-73.62, 36.47, 0.34) mm, rotated rx 180 ry 0 rz 90 deg; joints [74.328, -19.286, 90.457, 0, 18.829, 74.328]
  MoveL 1508 to (-75.13, 36.29, -0.06) mm, rotated rx 180 ry 0 rz 90 deg; joints [74.307, -19.286, 90.541, 0, 18.745, 74.307]
  MoveL 1509 to (-76.57, 35.78, -0.47) mm, rotated rx -180 ry 0 rz 90 deg; joints [74.276, -19.283, 90.613, 0, 18.67, 74.276]
  MoveL 1510 to (-77.85, 34.96, -0.87) mm, rotated rx -180 ry 0 rz 90 deg; joints [74.236, -19.277, 90.669, 0, 18.608, 74.236]
  MoveL 1511 to (-78.92, 33.88, -1.28) mm, rotated rx 180 ry 0 rz 90 deg; joints [74.189, -19.267, 90.706, 0, 18.561, 74.189]
  MoveL 1512 to (-79.72, 32.59, -1.69) mm, rotated rx 180 ry 0 rz 90 deg; joints [74.137, -19.252, 90.722, 0, 18.53, 74.137]
  MoveL 1513 to (-80.22, 31.16, -2.09) mm, rotated rx 180 ry 0 rz 90 deg; joints [74.083, -19.232, 90.714, 0, 18.518, 74.083]
  MoveL 1514 to (-80.36, 29.64, -2.5) mm, rotated rx 180 ry 0 rz 90 deg; joints [74.03, -19.206, 90.681, 0, 18.525, 74.03]
  MoveL 1515 to (-80.36, 0.47, -2.5) mm, rotated rx 180 ry 0 rz 90 deg; joints [73.041, -19.081, 90.108, 0, 18.973, 73.041]
  MoveC 1516 to (-78.13, -5.38, -2.5) mm, rotated rx 180 ry 0 rz 90 deg; joints [72.867, -19.021, 89.84, 0, 19.181, 72.867] to (-72.49, -8.11, -2.5) mm, rotated rx 180 ry 0 rz 90 deg; joints [72.834, -18.923, 89.407, 0, 19.516, 72.834]
  MoveL 1517 to (-72.02, -8.13, -2.5) mm, rotated rx -180 ry 0 rz 90 deg; joints [72.838, -18.916, 89.375, 0, 19.541, 72.838]
  MoveC 1518 to (-70.49, -8.09, -2.5) mm, rotated rx 180 ry 0 rz 90 deg; joints [72.856, -18.893, 89.273, 0, 19.62, 72.856] to (-68.97, -7.84, -2.5) mm, rotated rx -180 ry 0 rz 90 deg; joints [72.879, -18.871, 89.176, 0, 19.695, 72.879]
  MoveL 1519 to (-19.43, 3.56, -2.5) mm, rotated rx 180 ry 0 rz 90 deg; joints [73.747, -18.113, 86.02, 0, 22.093, 73.747]
  MoveC 1520 to (-13.88, 7.76, -2.5) mm, rotated rx -180 ry 0 rz 90 deg; joints [73.937, -18.037, 85.717, 0, 22.32, 73.937] to (-13.26, 14.69, -2.5) mm, rotated rx -180 ry 0 rz 90 deg; joints [74.169, -18.061, 85.812, 0, 22.249, 74.169]
  MoveL 1521 to (-13.58, 15.64, -2.5) mm, rotated rx 180 ry 0 rz 90 deg; joints [74.197, -18.071, 85.854, 0, 22.218, 74.197]
  MoveL 1522 to (-20.17, 34.04, -2.5) mm, rotated rx 180 ry 0 rz 90 deg; joints [74.742, -18.275, 86.67, 0, 21.605, 74.742]
  MoveC 1523 to (-21.63, 36.68, -2.5) mm, rotated rx 180 ry 0 rz 90 deg; joints [74.816, -18.312, 86.822, 0, 21.49, 74.816] to (-23.87, 38.7, -2.5) mm, rotated rx 180 ry 0 rz 90 deg; joints [74.863, -18.36, 87.016, 0, 21.344, 74.863]
  MoveL 1524 to (-66.23, 65.86, -2.5) mm, rotated rx -180 ry 0 rz 90 deg; joints [75.399, -19.145, 90.398, 0, 18.746, 75.399]
  MoveC 1525 to (-69.05, 67.21, -2.5) mm, rotated rx 180 ry 0 rz 90 deg; joints [75.42, -19.191, 90.611, 0, 18.58, 75.42] to (-72.13, 67.77, -2.5) mm, rotated rx 180 ry 0 rz 90 deg; joints [75.412, -19.238, 90.827, 0, 18.411, 75.412]
  MoveC 1526 to (-76.69, 66.52, -2.5) mm, rotated rx -180 ry 0 rz 90 deg; joints [75.328, -19.299, 91.109, 0, 18.189, 75.328] to (-79.62, 62.81, -2.5) mm, rotated rx -180 ry 0 rz 90 deg; joints [75.173, -19.326, 91.24, 0, 18.087, 75.173]
  MoveC 1527 to (-80.18, 60.77, -2.5) mm, rotated rx -180 ry 0 rz 90 deg; joints [75.098, -19.327, 91.24, 0, 18.086, 75.098] to (-80.36, 58.67, -2.5) mm, rotated rx 180 ry 0 rz 90 deg; joints [75.024, -19.321, 91.215, 0, 18.106, 75.024]
  MoveL 1528 to (-80.36, 29.64, -2.5) mm, rotated rx 180 ry 0 rz 90 deg; joints [74.03, -19.206, 90.681, 0, 18.525, 74.03]
  MoveL 1529 to (-72.81, 29.65, -2.5) mm, rotated rx 180 ry 0 rz 90 deg; joints [74.104, -19.096, 90.178, 0, 18.918, 74.104]
  MoveL 1530 to (-72.81, 29.65, 0.5) mm, rotated rx -180 ry 0 rz 90 deg; joints [74.104, -19.253, 90.279, 0, 18.975, 74.104]
  Establecer velocidad (1000.0 mm/s)
  MoveL 1531 to (-72.81, 29.65, 10) mm, rotated rx -180 ry 0 rz 90 deg; joints [74.104, -19.751, 90.595, 0, 19.157, 74.104]
  Establecer velocidad (66.7 mm/s)
  MoveL 1532 to (-72.12, -45.33, 10) mm, rotated rx 180 ry 0 rz 90 deg; joints [71.6, -19.384, 88.998, 0, 20.386, 71.6]
  MoveL 1533 to (-72.12, -45.33, 0.75) mm, rotated rx 180 ry 0 rz 90 deg; joints [71.6, -18.903, 88.691, 0, 20.212, 71.6]
  MoveL 1534 to (-73.63, -45.15, 0.34) mm, rotated rx 180 ry 0 rz 90 deg; joints [71.59, -18.906, 88.782, 0, 20.124, 71.59]
  MoveL 1535 to (-75.14, -45.33, -0.06) mm, rotated rx 180 ry 0 rz 90 deg; joints [71.567, -18.907, 88.865, 0, 20.042, 71.567]
  MoveL 1536 to (-76.57, -45.84, -0.47) mm, rotated rx 180 ry 0 rz 90 deg; joints [71.535, -18.906, 88.936, 0, 19.97, 71.535]
  MoveL 1537 to (-77.85, -46.66, -0.87) mm, rotated rx 180 ry 0 rz 90 deg; joints [71.493, -18.9, 88.99, 0, 19.91, 71.493]
  MoveL 1538 to (-78.92, -47.74, -1.28) mm, rotated rx 180 ry 0 rz 90 deg; joints [71.446, -18.89, 89.024, 0, 19.866, 71.446]
  MoveL 1539 to (-79.72, -49.02, -1.69) mm, rotated rx 180 ry 0 rz 90 deg; joints [71.394, -18.875, 89.035, 0, 19.84, 71.394]
  MoveL 1540 to (-80.22, -50.46, -2.09) mm, rotated rx -180 ry 0 rz 90 deg; joints [71.341, -18.854, 89.022, 0, 19.831, 71.341]
  MoveL 1541 to (-80.36, -51.97, -2.5) mm, rotated rx -180 ry 0 rz 90 deg; joints [71.29, -18.827, 88.984, 0, 19.843, 71.29]
  MoveL 1542 to (-80.36, -70.6, -2.5) mm, rotated rx 180 ry 0 rz 90 deg; joints [70.676, -18.727, 88.555, 0, 20.172, 70.676]
  MoveL 1543 to (-80.32, -71.55, -2.5) mm, rotated rx 180 ry 0 rz 90 deg; joints [70.645, -18.722, 88.531, 0, 20.191, 70.645]
  MoveC 1544 to (-77.55, -77.37, -2.5) mm, rotated rx -180 ry 0 rz 90 deg; joints [70.486, -18.646, 88.208, 0, 20.438, 70.486] to (-71.55, -79.73, -2.5) mm, rotated rx 180 ry 0 rz 90 deg; joints [70.479, -18.537, 87.749, 0, 20.788, 70.479]
  MoveL 1545 to (-70.6, -79.73, -2.5) mm, rotated rx -180 ry 0 rz 90 deg; joints [70.49, -18.522, 87.686, 0, 20.836, 70.49]
  MoveL 1546 to (-36.48, -79.45, -2.5) mm, rotated rx 180 ry 0 rz 90 deg; joints [70.885, -17.948, 85.366, 0, 22.582, 70.885]
  MoveL 1547 to (-35.25, -79.44, -2.5) mm, rotated rx -180 ry 0 rz 90 deg; joints [70.899, -17.926, 85.281, 0, 22.645, 70.899]
  MoveC 1548 to (-29.85, -77.53, -2.5) mm, rotated rx -180 ry 0 rz 90 deg; joints [71.019, -17.841, 84.952, 0, 22.889, 71.019] to (-26.71, -72.74, -2.5) mm, rotated rx 180 ry 0 rz 90 deg; joints [71.207, -17.814, 84.848, 0, 22.967, 71.207]
  MoveL 1549 to (-14.07, -24.17, -2.5) mm, rotated rx -180 ry 0 rz 90 deg; joints [72.898, -17.87, 85.064, 0, 22.806, 72.898]
  MoveC 1550 to (-13.81, -20.28, -2.5) mm, rotated rx -180 ry 0 rz 90 deg; joints [73.027, -17.887, 85.129, 0, 22.758, 73.027] to (-15.04, -16.58, -2.5) mm, rotated rx -180 ry 0 rz 90 deg; joints [73.134, -17.929, 85.295, 0, 22.635, 73.134]
  MoveC 1551 to (-18.62, -13.65, -2.5) mm, rotated rx -180 ry 0 rz 90 deg; joints [73.194, -18.009, 85.607, 0, 22.402, 73.194] to (-23.22, -13.12, -2.5) mm, rotated rx 180 ry 0 rz 90 deg; joints [73.166, -18.093, 85.939, 0, 22.154, 73.166]
  MoveL 1552 to (-24.17, -13.28, -2.5) mm, rotated rx 180 ry 0 rz 90 deg; joints [73.152, -18.108, 86.001, 0, 22.107, 73.152]
  MoveL 1553 to (-73.35, -23.74, -2.5) mm, rotated rx -180 ry 0 rz 90 deg; joints [72.303, -18.862, 89.136, 0, 19.726, 72.303]
  MoveC 1554 to (-78.39, -26.82, -2.5) mm, rotated rx 180 ry 0 rz 90 deg; joints [72.146, -18.923, 89.406, 0, 19.517, 72.146] to (-80.36, -32.39, -2.5) mm, rotated rx -180 ry 0 rz 90 deg; joints [71.939, -18.926, 89.417, 0, 19.508, 71.939]
  MoveL 1555 to (-80.36, -51.97, -2.5) mm, rotated rx -180 ry 0 rz 90 deg; joints [71.29, -18.827, 88.984, 0, 19.843, 71.29]
  MoveL 1556 to (-72.81, -51.97, -2.5) mm, rotated rx -180 ry 0 rz 90 deg; joints [71.374, -18.71, 88.479, 0, 20.231, 71.374]
  MoveL 1557 to (-72.81, -51.97, 0.5) mm, rotated rx 180 ry 0 rz 90 deg; joints [71.374, -18.865, 88.579, 0, 20.286, 71.374]
  Establecer velocidad (1000.0 mm/s)
  MoveL 1558 to (-72.81, -51.97, 10) mm, rotated rx -180 ry 0 rz 90 deg; joints [71.374, -19.359, 88.895, 0, 20.464, 71.374]
  Establecer velocidad (66.7 mm/s)
  MoveL 1559 to (18.62, -71.21, 10) mm, rotated rx -180 ry 0 rz 90 deg; joints [71.735, -17.592, 82.084, 0, 25.508, 71.735]
  MoveL 1560 to (18.62, -71.21, 0.75) mm, rotated rx 180 ry 0 rz 90 deg; joints [71.735, -17.125, 81.776, 0, 25.349, 71.735]
  MoveL 1561 to (18.45, -72.72, 0.34) mm, rotated rx 180 ry 0 rz 90 deg; joints [71.686, -17.097, 81.738, 0, 25.359, 71.686]
  MoveL 1562 to (18.65, -74.23, -0.06) mm, rotated rx -180 ry 0 rz 90 deg; joints [71.641, -17.063, 81.674, 0, 25.389, 71.641]
  MoveL 1563 to (19.17, -75.65, -0.47) mm, rotated rx 180 ry 0 rz 90 deg; joints [71.602, -17.022, 81.588, 0, 25.434, 71.602]
  MoveL 1564 to (20, -76.93, -0.87) mm, rotated rx 180 ry 0 rz 90 deg; joints [71.571, -16.976, 81.483, 0, 25.493, 71.571]
  MoveL 1565 to (21.09, -77.99, -1.28) mm, rotated rx 180 ry 0 rz 90 deg; joints [71.549, -16.926, 81.365, 0, 25.561, 71.549]
  MoveL 1566 to (22.39, -78.78, -1.69) mm, rotated rx 180 ry 0 rz 90 deg; joints [71.538, -16.874, 81.238, 0, 25.636, 71.538]
  MoveL 1567 to (23.83, -79.26, -2.09) mm, rotated rx 180 ry 0 rz 90 deg; joints [71.538, -16.821, 81.108, 0, 25.713, 71.538]
  MoveL 1568 to (25.34, -79.39, -2.5) mm, rotated rx 180 ry 0 rz 90 deg; joints [71.55, -16.769, 80.981, 0, 25.788, 71.55]
  MoveL 1569 to (45.96, -79.17, -2.5) mm, rotated rx -180 ry 0 rz 90 deg; joints [71.767, -16.336, 79.47, 0, 26.866, 71.767]
  MoveL 1570 to (53.54, -79.07, -2.5) mm, rotated rx 180 ry 0 rz 90 deg; joints [71.847, -16.173, 78.908, 0, 27.264, 71.847]
  MoveC 1571 to (55.25, -78.94, -2.5) mm, rotated rx 180 ry 0 rz 90 deg; joints [71.868, -16.136, 78.784, 0, 27.352, 71.868] to (56.91, -78.55, -2.5) mm, rotated rx 180 ry 0 rz 90 deg; joints [71.897, -16.102, 78.669, 0, 27.433, 71.897]
  MoveC 1572 to (60.85, -74.88, -2.5) mm, rotated rx 180 ry 0 rz 90 deg; joints [72.048, -16.041, 78.463, 0, 27.579, 72.048] to (60.51, -69.49, -2.5) mm, rotated rx 180 ry 0 rz 90 deg; joints [72.21, -16.088, 78.619, 0, 27.468, 72.21]
  MoveL 1573 to (60.41, -69.31, -2.5) mm, rotated rx 180 ry 0 rz 90 deg; joints [72.215, -16.091, 78.631, 0, 27.46, 72.215]
  MoveC 1574 to (59.46, -67.8, -2.5) mm, rotated rx -180 ry 0 rz 90 deg; joints [72.252, -16.123, 78.738, 0, 27.384, 72.252] to (58.37, -66.39, -2.5) mm, rotated rx -180 ry 0 rz 90 deg; joints [72.284, -16.157, 78.854, 0, 27.303, 72.284]
  MoveL 1575 to (29.85, -33.42, -2.5) mm, rotated rx -180 ry 0 rz 90 deg; joints [73.032, -16.976, 81.722, 0, 25.254, 73.032]
  MoveL 1576 to (29.19, -32.69, -2.5) mm, rotated rx 180 ry 0 rz 90 deg; joints [73.049, -16.994, 81.786, 0, 25.208, 73.049]
  MoveL 1577 to (28.9, -32.42, -2.5) mm, rotated rx 180 ry 0 rz 90 deg; joints [73.055, -17.001, 81.813, 0, 25.188, 73.055]
  MoveL 1578 to (14.69, -21.03, -2.5) mm, rotated rx 180 ry 0 rz 90 deg; joints [73.279, -17.35, 83.09, 0, 24.26, 73.279]
  MoveL 1579 to (13.82, -20.37, -2.5) mm, rotated rx -180 ry 0 rz 90 deg; joints [73.292, -17.371, 83.166, 0, 24.204, 73.292]
  MoveC 1580 to (11.55, -19.06, -2.5) mm, rotated rx 180 ry 0 rz 90 deg; joints [73.312, -17.422, 83.358, 0, 24.064, 73.312] to (9, -18.39, -2.5) mm, rotated rx 180 ry 0 rz 90 deg; joints [73.309, -17.475, 83.554, 0, 23.92, 73.309]
  MoveC 1581 to (5.5, -18.99, -2.5) mm, rotated rx -180 ry 0 rz 90 deg; joints [73.256, -17.538, 83.791, 0, 23.746, 73.256] to (2.83, -21.33, -2.5) mm, rotated rx 180 ry 0 rz 90 deg; joints [73.155, -17.575, 83.931, 0, 23.644, 73.155]
  MoveC 1582 to (1.99, -22.89, -2.5) mm, rotated rx -180 ry 0 rz 90 deg; joints [73.097, -17.582, 83.957, 0, 23.624, 73.097] to (1.4, -24.56, -2.5) mm, rotated rx 180 ry 0 rz 90 deg; joints [73.038, -17.583, 83.963, 0, 23.62, 73.038]
  MoveL 1583 to (-10.7, -70.14, -2.5) mm, rotated rx 180 ry 0 rz 90 deg; joints [71.461, -17.536, 83.787, 0, 23.75, 71.461]
  MoveC 1584 to (-10.76, -73.9, -2.5) mm, rotated rx 180 ry 0 rz 90 deg; joints [71.342, -17.514, 83.701, 0, 23.812, 71.342] to (-9.03, -77.23, -2.5) mm, rotated rx 180 ry 0 rz 90 deg; joints [71.255, -17.46, 83.5, 0, 23.96, 71.255]
  MoveC 1585 to (-6.18, -79.06, -2.5) mm, rotated rx -180 ry 0 rz 90 deg; joints [71.228, -17.394, 83.254, 0, 24.14, 71.228] to (-2.86, -79.67, -2.5) mm, rotated rx -180 ry 0 rz 90 deg; joints [71.244, -17.327, 83.003, 0, 24.323, 71.244]
  MoveL 1586 to (25.34, -79.39, -2.5) mm, rotated rx 180 ry 0 rz 90 deg; joints [71.55, -16.769, 80.981, 0, 25.788, 71.55]
  MoveL 1587 to (25.27, -71.84, -2.5) mm, rotated rx -180 ry 0 rz 90 deg; joints [71.784, -16.821, 81.169, 0, 25.653, 71.784]
  MoveL 1588 to (25.27, -71.84, 0.5) mm, rotated rx 180 ry 0 rz 90 deg; joints [71.784, -16.973, 81.27, 0, 25.703, 71.784]
  Establecer velocidad (1000.0 mm/s)
  MoveL 1589 to (25.27, -71.84, 10) mm, rotated rx 180 ry 0 rz 90 deg; joints [71.784, -17.452, 81.587, 0, 25.865, 71.784]
  Establecer velocidad (66.7 mm/s)
  MoveL 1590 to (69.68, -28.72, 10) mm, rotated rx 180 ry 0 rz 90 deg; joints [73.552, -16.788, 79.295, 0, 27.493, 73.552]
  MoveL 1591 to (69.68, -28.72, 0.75) mm, rotated rx 180 ry 0 rz 90 deg; joints [73.552, -16.325, 78.984, 0, 27.341, 73.552]
  MoveL 1592 to (71.18, -28.91, 0.34) mm, rotated rx 180 ry 0 rz 90 deg; joints [73.56, -16.27, 78.853, 0, 27.417, 73.56]
  MoveL 1593 to (72.69, -28.72, -0.06) mm, rotated rx 180 ry 0 rz 90 deg; joints [73.579, -16.218, 78.729, 0, 27.488, 73.579]
  MoveL 1594 to (74.12, -28.21, -0.47) mm, rotated rx 180 ry 0 rz 90 deg; joints [73.608, -16.169, 78.619, 0, 27.55, 73.608]
  MoveL 1595 to (75.4, -27.4, -0.87) mm, rotated rx 180 ry 0 rz 90 deg; joints [73.645, -16.125, 78.526, 0, 27.599, 73.645]
  MoveL 1596 to (76.47, -26.32, -1.28) mm, rotated rx 180 ry 0 rz 90 deg; joints [73.688, -16.088, 78.455, 0, 27.633, 73.688]
  MoveL 1597 to (77.28, -25.03, -1.69) mm, rotated rx -180 ry 0 rz 90 deg; joints [73.735, -16.058, 78.409, 0, 27.649, 73.735]
  MoveL 1598 to (77.78, -23.59, -2.09) mm, rotated rx -180 ry 0 rz 90 deg; joints [73.784, -16.036, 78.389, 0, 27.647, 73.784]
  MoveL 1599 to (77.92, -22.08, -2.5) mm, rotated rx 180 ry 0 rz 90 deg; joints [73.832, -16.022, 78.398, 0, 27.625, 73.832]
  MoveL 1600 to (77.92, -5.21, -2.5) mm, rotated rx -180 ry 0 rz 90 deg; joints [74.354, -16.13, 78.762, 0, 27.367, 74.354]
  MoveC 1601 to (77.83, -2.83, -2.5) mm, rotated rx 180 ry 0 rz 90 deg; joints [74.427, -16.147, 78.819, 0, 27.327, 74.427] to (77.51, -0.47, -2.5) mm, rotated rx 180 ry 0 rz 90 deg; joints [74.497, -16.168, 78.894, 0, 27.275, 74.497]
  MoveC 1602 to (73.8, 3.55, -2.5) mm, rotated rx -180 ry 0 rz 90 deg; joints [74.591, -16.275, 79.258, 0, 27.017, 74.591] to (68.33, 3.57, -2.5) mm, rotated rx -180 ry 0 rz 90 deg; joints [74.544, -16.395, 79.671, 0, 26.724, 74.544]
  MoveC 1603 to (66.84, 2.21, -2.5) mm, rotated rx -180 ry 0 rz 90 deg; joints [74.489, -16.419, 79.754, 0, 26.664, 74.489] to (65.55, 0.68, -2.5) mm, rotated rx -180 ry 0 rz 90 deg; joints [74.429, -16.437, 79.819, 0, 26.618, 74.429]
  MoveL 1604 to (62.61, -3.32, -2.5) mm, rotated rx -180 ry 0 rz 90 deg; joints [74.279, -16.476, 79.955, 0, 26.521, 74.279]
  MoveL 1605 to (49.49, -21.32, -2.5) mm, rotated rx -180 ry 0 rz 90 deg; joints [73.597, -16.645, 80.546, 0, 26.1, 73.597]
  MoveL 1606 to (48.9, -22.2, -2.5) mm, rotated rx 180 ry 0 rz 90 deg; joints [73.564, -16.652, 80.571, 0, 26.082, 73.564]
  MoveC 1607 to (47.72, -26.49, -2.5) mm, rotated rx 180 ry 0 rz 90 deg; joints [73.419, -16.65, 80.564, 0, 26.087, 73.419] to (49.42, -30.6, -2.5) mm, rotated rx -180 ry 0 rz 90 deg; joints [73.306, -16.589, 80.347, 0, 26.242, 73.306]
  MoveL 1608 to (52.1, -33.64, -2.5) mm, rotated rx -180 ry 0 rz 90 deg; joints [73.237, -16.512, 80.08, 0, 26.432, 73.237]
  MoveL 1609 to (65.52, -48.8, -2.5) mm, rotated rx -180 ry 0 rz 90 deg; joints [72.894, -16.121, 78.731, 0, 27.39, 72.894]
  MoveL 1610 to (66.41, -49.75, -2.5) mm, rotated rx 180 ry 0 rz 90 deg; joints [72.873, -16.094, 78.642, 0, 27.452, 72.873]
  MoveC 1611 to (67.9, -51.07, -2.5) mm, rotated rx -180 ry 0 rz 90 deg; joints [72.847, -16.052, 78.499, 0, 27.553, 72.847] to (69.65, -52.01, -2.5) mm, rotated rx -180 ry 0 rz 90 deg; joints [72.834, -16.007, 78.345, 0, 27.662, 72.834]
  MoveC 1612 to (74.28, -51.35, -2.5) mm, rotated rx 180 ry 0 rz 90 deg; joints [72.898, -15.907, 78.01, 0, 27.897, 72.898] to (77.38, -47.86, -2.5) mm, rotated rx 180 ry 0 rz 90 deg; joints [73.034, -15.861, 77.855, 0, 28.006, 73.034]
  MoveC 1613 to (77.78, -45.8, -2.5) mm, rotated rx -180 ry 0 rz 90 deg; joints [73.101, -15.866, 77.872, 0, 27.994, 73.101] to (77.92, -43.72, -2.5) mm, rotated rx -180 ry 0 rz 90 deg; joints [73.166, -15.877, 77.91, 0, 27.967, 73.166]
  MoveL 1614 to (77.92, -22.08, -2.5) mm, rotated rx 180 ry 0 rz 90 deg; joints [73.832, -16.022, 78.398, 0, 27.625, 73.832]
  MoveL 1615 to (70.37, -22.08, -2.5) mm, rotated rx 180 ry 0 rz 90 deg; joints [73.764, -16.19, 78.969, 0, 27.221, 73.764]
  MoveL 1616 to (70.37, -22.08, 0.5) mm, rotated rx 180 ry 0 rz 90 deg; joints [73.764, -16.341, 79.071, 0, 27.27, 73.764]
  Establecer velocidad (1000.0 mm/s)
  MoveL 1617 to (70.37, -22.08, 10) mm, rotated rx 180 ry 0 rz 90 deg; joints [73.764, -16.816, 79.39, 0, 27.427, 73.764]
  Establecer velocidad (66.7 mm/s)
  MoveL 1618 to (38.79, 26.98, 10) mm, rotated rx -180 ry 0 rz 90 deg; joints [75.03, -17.777, 82.748, 0, 25.028, 75.03]
  MoveL 1619 to (38.79, 26.98, 0.75) mm, rotated rx 180 ry 0 rz 90 deg; joints [75.03, -17.308, 82.44, 0, 24.868, 75.03]
  MoveL 1620 to (38.93, 28.49, 0.34) mm, rotated rx -180 ry 0 rz 90 deg; joints [75.079, -17.293, 82.445, 0, 24.848, 75.079]
  MoveL 1621 to (38.71, 29.99, -0.06) mm, rotated rx -180 ry 0 rz 90 deg; joints [75.126, -17.285, 82.477, 0, 24.808, 75.126]
  MoveL 1622 to (38.16, 31.41, -0.47) mm, rotated rx 180 ry 0 rz 90 deg; joints [75.166, -17.283, 82.531, 0, 24.752, 75.166]
  MoveL 1623 to (37.31, 32.67, -0.87) mm, rotated rx 180 ry 0 rz 90 deg; joints [75.199, -17.286, 82.604, 0, 24.682, 75.199]
  MoveL 1624 to (36.2, 33.71, -1.28) mm, rotated rx 180 ry 0 rz 90 deg; joints [75.223, -17.293, 82.691, 0, 24.602, 75.223]
  MoveL 1625 to (34.89, 34.48, -1.69) mm, rotated rx -180 ry 0 rz 90 deg; joints [75.237, -17.302, 82.788, 0, 24.514, 75.237]
  MoveL 1626 to (33.44, 34.94, -2.09) mm, rotated rx 180 ry 0 rz 90 deg; joints [75.239, -17.312, 82.888, 0, 24.424, 75.239]
  MoveL 1627 to (31.93, 35.03, -2.5) mm, rotated rx -180 ry 0 rz 90 deg; joints [75.23, -17.322, 82.986, 0, 24.336, 75.23]
  MoveL 1628 to (8.05, 34.39, -2.5) mm, rotated rx -180 ry 0 rz 90 deg; joints [75.004, -17.774, 84.691, 0, 23.083, 75.004]
  MoveL 1629 to (7.11, 34.33, -2.5) mm, rotated rx -180 ry 0 rz 90 deg; joints [74.994, -17.791, 84.757, 0, 23.034, 74.994]
  MoveC 1630 to (3.57, 33.31, -2.5) mm, rotated rx 180 ry 0 rz 90 deg; joints [74.929, -17.851, 84.989, 0, 22.862, 74.929] to (0.87, 30.8, -2.5) mm, rotated rx -180 ry 0 rz 90 deg; joints [74.823, -17.888, 85.132, 0, 22.756, 74.823]
  MoveC 1631 to (0, 28.04, -2.5) mm, rotated rx 180 ry 0 rz 90 deg; joints [74.726, -17.89, 85.14, 0, 22.749, 74.726] to (0.25, 25.16, -2.5) mm, rotated rx 180 ry 0 rz 90 deg; joints [74.634, -17.871, 85.067, 0, 22.804, 74.634]
  MoveL 1632 to (0.54, 24.17, -2.5) mm, rotated rx -180 ry 0 rz 90 deg; joints [74.604, -17.861, 85.027, 0, 22.834, 74.604]
  MoveL 1633 to (6.38, 8.05, -2.5) mm, rotated rx -180 ry 0 rz 90 deg; joints [74.135, -17.67, 84.292, 0, 23.378, 74.135]
  MoveL 1634 to (6.73, 7.11, -2.5) mm, rotated rx 180 ry 0 rz 90 deg; joints [74.107, -17.658, 84.248, 0, 23.41, 74.107]
  MoveC 1635 to (7.66, 5.39, -2.5) mm, rotated rx 180 ry 0 rz 90 deg; joints [74.06, -17.632, 84.147, 0, 23.485, 74.06] to (9, 3.97, -2.5) mm, rotated rx 180 ry 0 rz 90 deg; joints [74.027, -17.599, 84.022, 0, 23.576, 74.027]
  MoveL 1636 to (9.95, 3.21, -2.5) mm, rotated rx 180 ry 0 rz 90 deg; joints [74.011, -17.577, 83.939, 0, 23.638, 74.011]
  MoveL 1637 to (26.06, -9.32, -2.5) mm, rotated rx 180 ry 0 rz 90 deg; joints [73.759, -17.195, 82.519, 0, 24.676, 73.759]
  MoveL 1638 to (26.92, -9.95, -2.5) mm, rotated rx 180 ry 0 rz 90 deg; joints [73.747, -17.175, 82.443, 0, 24.731, 73.747]
  MoveC 1639 to (31.93, -11.22, -2.5) mm, rotated rx -180 ry 0 rz 90 deg; joints [73.753, -17.067, 82.053, 0, 25.015, 73.753] to (36.48, -8.78, -2.5) mm, rotated rx 180 ry 0 rz 90 deg; joints [73.872, -16.99, 81.772, 0, 25.218, 73.872]
  MoveL 1640 to (37.12, -8.05, -2.5) mm, rotated rx -180 ry 0 rz 90 deg; joints [73.901, -16.981, 81.74, 0, 25.24, 73.901]
  MoveL 1641 to (40.27, -3.69, -2.5) mm, rotated rx -180 ry 0 rz 90 deg; joints [74.068, -16.942, 81.602, 0, 25.341, 74.068]
  MoveL 1642 to (57.33, 20.07, -2.5) mm, rotated rx -180 ry 0 rz 90 deg; joints [74.968, -16.725, 80.828, 0, 25.897, 74.968]
  MoveL 1643 to (59.9, 23.65, -2.5) mm, rotated rx 180 ry 0 rz 90 deg; joints [75.103, -16.692, 80.709, 0, 25.983, 75.103]
  MoveC 1644 to (60.89, 25.25, -2.5) mm, rotated rx 180 ry 0 rz 90 deg; joints [75.162, -16.68, 80.666, 0, 26.013, 75.162] to (61.67, 26.96, -2.5) mm, rotated rx -180 ry 0 rz 90 deg; joints [75.222, -16.673, 80.642, 0, 26.031, 75.222]
  MoveC 1645 to (61.23, 32.36, -2.5) mm, rotated rx 180 ry 0 rz 90 deg; joints [75.39, -16.712, 80.781, 0, 25.931, 75.39] to (56.75, 35.42, -2.5) mm, rotated rx -180 ry 0 rz 90 deg; joints [75.45, -16.822, 81.173, 0, 25.65, 75.45]
  MoveC 1646 to (55.15, 35.59, -2.5) mm, rotated rx 180 ry 0 rz 90 deg; joints [75.442, -16.857, 81.294, 0, 25.562, 75.442] to (53.54, 35.61, -2.5) mm, rotated rx 180 ry 0 rz 90 deg; joints [75.429, -16.89, 81.413, 0, 25.476, 75.429]
  MoveL 1647 to (51.65, 35.57, -2.5) mm, rotated rx -180 ry 0 rz 90 deg; joints [75.412, -16.929, 81.553, 0, 25.376, 75.412]
  MoveL 1648 to (31.93, 35.03, -2.5) mm, rotated rx -180 ry 0 rz 90 deg; joints [75.23, -17.322, 82.986, 0, 24.336, 75.23]
  MoveL 1649 to (32.13, 27.49, -2.5) mm, rotated rx -180 ry 0 rz 90 deg; joints [74.989, -17.279, 82.826, 0, 24.453, 74.989]
  MoveL 1650 to (32.13, 27.49, 0.5) mm, rotated rx 180 ry 0 rz 90 deg; joints [74.989, -17.431, 82.927, 0, 24.504, 74.989]
  Establecer velocidad (1000.0 mm/s)
  MoveL 1651 to (32.13, 27.49, 10) mm, rotated rx -180 ry 0 rz 90 deg; joints [74.989, -17.913, 83.243, 0, 24.67, 74.989]
  Establecer velocidad (66.7 mm/s)
  MoveL 1652 to (27.37, 70.93, 10) mm, rotated rx 180 ry 0 rz 90 deg; joints [76.354, -18.223, 84.391, 0, 23.832, 76.354]
  MoveL 1653 to (27.37, 70.93, 0.75) mm, rotated rx 180 ry 0 rz 90 deg; joints [76.354, -17.752, 84.083, 0, 23.668, 76.354]
  MoveL 1654 to (27.58, 72.43, 0.34) mm, rotated rx 180 ry 0 rz 90 deg; joints [76.404, -17.734, 84.081, 0, 23.653, 76.404]
  MoveL 1655 to (27.42, 73.94, -0.06) mm, rotated rx 180 ry 0 rz 90 deg; joints [76.452, -17.723, 84.105, 0, 23.618, 76.452]
  MoveL 1656 to (26.93, 75.38, -0.47) mm, rotated rx -180 ry 0 rz 90 deg; joints [76.495, -17.719, 84.152, 0, 23.566, 76.495]
  MoveL 1657 to (26.13, 76.67, -0.87) mm, rotated rx 180 ry 0 rz 90 deg; joints [76.531, -17.719, 84.219, 0, 23.5, 76.531]
  MoveL 1658 to (25.06, 77.76, -1.28) mm, rotated rx 180 ry 0 rz 90 deg; joints [76.558, -17.723, 84.3, 0, 23.423, 76.558]
  MoveL 1659 to (23.79, 78.58, -1.69) mm, rotated rx 180 ry 0 rz 90 deg; joints [76.575, -17.73, 84.393, 0, 23.338, 76.575]
  MoveL 1660 to (22.36, 79.1, -2.09) mm, rotated rx 180 ry 0 rz 90 deg; joints [76.581, -17.739, 84.491, 0, 23.248, 76.581]
  MoveL 1661 to (20.85, 79.26, -2.5) mm, rotated rx -180 ry 0 rz 90 deg; joints [76.574, -17.747, 84.588, 0, 23.159, 76.574]
  MoveC 1662 to (-4.5, 79.57, -2.5) mm, rotated rx 180 ry 0 rz 90 deg; joints [76.384, -18.207, 86.394, 0, 21.812, 76.384] to (-29.85, 79.78, -2.5) mm, rotated rx -180 ry 0 rz 90 deg; joints [76.184, -18.635, 88.163, 0, 20.472, 76.184]
  MoveC 1663 to (-33.37, 79.61, -2.5) mm, rotated rx 180 ry 0 rz 90 deg; joints [76.149, -18.692, 88.403, 0, 20.289, 76.149] to (-36.84, 78.98, -2.5) mm, rotated rx -180 ry 0 rz 90 deg; joints [76.099, -18.745, 88.63, 0, 20.115, 76.099]
  MoveC 1664 to (-41.43, 74.35, -2.5) mm, rotated rx -180 ry 0 rz 90 deg; joints [75.904, -18.8, 88.866, 0, 19.934, 75.904] to (-39.48, 68.13, -2.5) mm, rotated rx -180 ry 0 rz 90 deg; joints [75.71, -18.744, 88.625, 0, 20.119, 75.71]
  MoveC 1665 to (-37.5, 66.51, -2.5) mm, rotated rx -180 ry 0 rz 90 deg; joints [75.673, -18.705, 88.461, 0, 20.245, 75.673] to (-35.4, 65.06, -2.5) mm, rotated rx 180 ry 0 rz 90 deg; joints [75.642, -18.666, 88.291, 0, 20.374, 75.642]
  MoveL 1666 to (-13.36, 51.1, -2.5) mm, rotated rx -180 ry 0 rz 90 deg; joints [75.366, -18.236, 86.513, 0, 21.723, 75.366]
  MoveC 1667 to (-10.12, 49.71, -2.5) mm, rotated rx -180 ry 0 rz 90 deg; joints [75.348, -18.174, 86.261, 0, 21.912, 75.348] to (-6.61, 49.42, -2.5) mm, rotated rx -180 ry 0 rz 90 deg; joints [75.369, -18.111, 86.01, 0, 22.101, 75.369]
  MoveC 1668 to (32.66, 52.31, -2.5) mm, rotated rx 180 ry 0 rz 90 deg; joints [75.792, -17.395, 83.258, 0, 24.138, 75.792] to (71.94, 55.04, -2.5) mm, rotated rx -180 ry 0 rz 90 deg; joints [76.193, -16.606, 80.409, 0, 26.198, 76.193]
  MoveC 1669 to (75.88, 56.91, -2.5) mm, rotated rx -180 ry 0 rz 90 deg; joints [76.283, -16.531, 80.147, 0, 26.385, 76.283] to (77.48, 60.97, -2.5) mm, rotated rx 180 ry 0 rz 90 deg; joints [76.423, -16.518, 80.101, 0, 26.418, 76.423]
  MoveL 1670 to (77.48, 71.55, -2.5) mm, rotated rx -180 ry 0 rz 90 deg; joints [76.758, -16.573, 80.291, 0, 26.282, 76.758]
  MoveL 1671 to (77.47, 72.49, -2.5) mm, rotated rx 180 ry 0 rz 90 deg; joints [76.788, -16.578, 80.308, 0, 26.269, 76.788]
  MoveC 1672 to (75.71, 76.64, -2.5) mm, rotated rx -180 ry 0 rz 90 deg; joints [76.907, -16.636, 80.513, 0, 26.123, 76.907] to (71.55, 78.34, -2.5) mm, rotated rx 180 ry 0 rz 90 deg; joints [76.93, -16.733, 80.856, 0, 25.877, 76.93]
  MoveC 1673 to (46.2, 78.85, -2.5) mm, rotated rx 180 ry 0 rz 90 deg; joints [76.757, -17.256, 82.743, 0, 24.513, 76.757] to (20.85, 79.26, -2.5) mm, rotated rx 180 ry 0 rz 90 deg; joints [76.574, -17.747, 84.588, 0, 23.159, 76.574]
  MoveL 1674 to (20.74, 71.71, -2.5) mm, rotated rx 180 ry 0 rz 90 deg; joints [76.327, -17.715, 84.465, 0, 23.25, 76.327]
  MoveL 1675 to (20.74, 71.71, 0.5) mm, rotated rx 180 ry 0 rz 90 deg; joints [76.327, -17.868, 84.566, 0, 23.302, 76.327]
  Establecer velocidad (1000.0 mm/s)
  MoveL 1676 to (20.74, 71.71, 10) mm, rotated rx 180 ry 0 rz 90 deg; joints [76.327, -18.353, 84.882, 0, 23.472, 76.327]
  Establecer velocidad (66.7 mm/s)
  MoveL 1677 to (27.39, 70.53, 10) mm, rotated rx -180 ry 0 rz 90 deg; joints [76.341, -18.221, 84.383, 0, 23.838, 76.341]
  MoveL 1678 to (27.39, 70.53, 0.5) mm, rotated rx 180 ry 0 rz 90 deg; joints [76.341, -17.737, 84.067, 0, 23.67, 76.341]
  MoveL 1679 to (27.59, 72.04, 0.09) mm, rotated rx 180 ry 0 rz 90 deg; joints [76.391, -17.719, 84.065, 0, 23.654, 76.391]
  MoveL 1680 to (27.43, 73.55, -0.31) mm, rotated rx -180 ry 0 rz 90 deg; joints [76.439, -17.709, 84.09, 0, 23.619, 76.439]
  MoveL 1681 to (26.93, 74.99, -0.72) mm, rotated rx 180 ry 0 rz 90 deg; joints [76.482, -17.704, 84.137, 0, 23.567, 76.482]
  MoveL 1682 to (26.13, 76.28, -1.13) mm, rotated rx 180 ry 0 rz 90 deg; joints [76.518, -17.704, 84.203, 0, 23.501, 76.518]
  MoveL 1683 to (25.06, 77.36, -1.53) mm, rotated rx 180 ry 0 rz 90 deg; joints [76.545, -17.709, 84.285, 0, 23.424, 76.545]
  MoveL 1684 to (23.78, 78.19, -1.94) mm, rotated rx 180 ry 0 rz 90 deg; joints [76.562, -17.716, 84.378, 0, 23.338, 76.562]
  MoveL 1685 to (22.35, 78.7, -2.34) mm, rotated rx 180 ry 0 rz 90 deg; joints [76.568, -17.724, 84.476, 0, 23.249, 76.568]
  MoveL 1686 to (20.85, 78.86, -2.75) mm, rotated rx 180 ry 0 rz 90 deg; joints [76.561, -17.732, 84.573, 0, 23.159, 76.561]
  MoveC 1687 to (15.87, 78.91, -2.75) mm, rotated rx -180 ry 0 rz 90 deg; joints [76.524, -17.825, 84.93, 0, 22.895, 76.524] to (10.9, 78.96, -2.75) mm, rotated rx 180 ry 0 rz 90 deg; joints [76.486, -17.916, 85.286, 0, 22.63, 76.486]
  MoveL 1688 to (-29.66, 79.38, -2.75) mm, rotated rx -180 ry 0 rz 90 deg; joints [76.172, -18.618, 88.135, 0, 20.483, 76.172]
  MoveC 1689 to (-32.61, 79.27, -2.75) mm, rotated rx 180 ry 0 rz 90 deg; joints [76.144, -18.665, 88.336, 0, 20.329, 76.144] to (-35.54, 78.87, -2.75) mm, rotated rx -180 ry 0 rz 90 deg; joints [76.106, -18.711, 88.531, 0, 20.18, 76.106]
  MoveL 1690 to (-36.48, 78.66, -2.75) mm, rotated rx -180 ry 0 rz 90 deg; joints [76.091, -18.725, 88.592, 0, 20.133, 76.091]
  MoveC 1691 to (-40.65, 74.79, -2.75) mm, rotated rx -180 ry 0 rz 90 deg; joints [75.925, -18.776, 88.811, 0, 19.965, 75.925] to (-39.88, 69.15, -2.75) mm, rotated rx 180 ry 0 rz 90 deg; joints [75.741, -18.741, 88.661, 0, 20.08, 75.741]
  MoveC 1692 to (-37.82, 67.25, -2.75) mm, rotated rx -180 ry 0 rz 90 deg; joints [75.695, -18.7, 88.487, 0, 20.213, 75.695] to (-35.54, 65.64, -2.75) mm, rotated rx -180 ry 0 rz 90 deg; joints [75.66, -18.657, 88.302, 0, 20.355, 75.66]
  MoveL 1693 to (-13.07, 51.4, -2.75) mm, rotated rx 180 ry 0 rz 90 deg; joints [75.379, -18.22, 86.49, 0, 21.729, 75.379]
  MoveC 1694 to (-10.03, 50.1, -2.75) mm, rotated rx -180 ry 0 rz 90 deg; joints [75.362, -18.161, 86.254, 0, 21.907, 75.362] to (-6.74, 49.82, -2.75) mm, rotated rx -180 ry 0 rz 90 deg; joints [75.381, -18.102, 86.017, 0, 22.084, 75.381]
  MoveC 1695 to (32.59, 52.7, -2.75) mm, rotated rx 180 ry 0 rz 90 deg; joints [75.805, -17.386, 83.261, 0, 24.125, 75.805] to (71.93, 55.47, -2.75) mm, rotated rx 180 ry 0 rz 90 deg; joints [76.206, -16.596, 80.409, 0, 26.187, 76.206]
  MoveC 1696 to (75.59, 57.21, -2.75) mm, rotated rx 180 ry 0 rz 90 deg; joints [76.29, -16.527, 80.166, 0, 26.361, 76.29] to (77.07, 60.98, -2.75) mm, rotated rx -180 ry 0 rz 90 deg; joints [76.42, -16.514, 80.123, 0, 26.392, 76.42]
  MoveL 1697 to (77.08, 71.55, -2.75) mm, rotated rx -180 ry 0 rz 90 deg; joints [76.755, -16.569, 80.313, 0, 26.256, 76.755]
  MoveL 1698 to (77.07, 72.49, -2.75) mm, rotated rx -180 ry 0 rz 90 deg; joints [76.785, -16.574, 80.33, 0, 26.244, 76.785]
  MoveC 1699 to (75.42, 76.35, -2.75) mm, rotated rx 180 ry 0 rz 90 deg; joints [76.895, -16.628, 80.522, 0, 26.107, 76.895] to (71.55, 77.94, -2.75) mm, rotated rx 180 ry 0 rz 90 deg; joints [76.918, -16.719, 80.84, 0, 25.878, 76.918]
  MoveC 1700 to (46.2, 78.48, -2.75) mm, rotated rx -180 ry 0 rz 90 deg; joints [76.744, -17.242, 82.728, 0, 24.514, 76.744] to (20.85, 78.86, -2.75) mm, rotated rx 180 ry 0 rz 90 deg; joints [76.561, -17.732, 84.573, 0, 23.159, 76.561]
  MoveL 1701 to (20.76, 71.31, -2.75) mm, rotated rx -180 ry 0 rz 90 deg; joints [76.314, -17.7, 84.449, 0, 23.251, 76.314]
  MoveL 1702 to (20.76, 71.31, 0.25) mm, rotated rx 180 ry 0 rz 90 deg; joints [76.314, -17.853, 84.55, 0, 23.304, 76.314]
  Establecer velocidad (1000.0 mm/s)
  MoveL 1703 to (20.76, 71.31, 10) mm, rotated rx 180 ry 0 rz 90 deg; joints [76.314, -18.351, 84.874, 0, 23.477, 76.314]
  Establecer velocidad (66.7 mm/s)
  MoveL 1704 to (38.71, 26.58, 10) mm, rotated rx 180 ry 0 rz 90 deg; joints [75.017, -17.776, 82.747, 0, 25.03, 75.017]
  MoveL 1705 to (38.71, 26.58, 0.5) mm, rotated rx -180 ry 0 rz 90 deg; joints [75.017, -17.295, 82.43, 0, 24.865, 75.017]
  MoveL 1706 to (38.85, 28.09, 0.09) mm, rotated rx 180 ry 0 rz 90 deg; joints [75.066, -17.28, 82.435, 0, 24.845, 75.066]
  MoveL 1707 to (38.63, 29.59, -0.31) mm, rotated rx -180 ry 0 rz 90 deg; joints [75.112, -17.272, 82.467, 0, 24.805, 75.112]
  MoveL 1708 to (38.08, 31.01, -0.72) mm, rotated rx -180 ry 0 rz 90 deg; joints [75.153, -17.27, 82.521, 0, 24.749, 75.153]
  MoveL 1709 to (37.23, 32.27, -1.13) mm, rotated rx 180 ry 0 rz 90 deg; joints [75.186, -17.273, 82.594, 0, 24.679, 75.186]
  MoveL 1710 to (36.12, 33.31, -1.53) mm, rotated rx 180 ry 0 rz 90 deg; joints [75.21, -17.28, 82.681, 0, 24.599, 75.21]
  MoveL 1711 to (34.81, 34.08, -1.94) mm, rotated rx 180 ry 0 rz 90 deg; joints [75.223, -17.289, 82.778, 0, 24.511, 75.223]
  MoveL 1712 to (33.36, 34.54, -2.34) mm, rotated rx -180 ry 0 rz 90 deg; joints [75.226, -17.299, 82.878, 0, 24.421, 75.226]
  MoveL 1713 to (31.85, 34.64, -2.75) mm, rotated rx 180 ry 0 rz 90 deg; joints [75.216, -17.309, 82.976, 0, 24.333, 75.216]
  MoveL 1714 to (10.9, 34.07, -2.75) mm, rotated rx 180 ry 0 rz 90 deg; joints [75.018, -17.706, 84.473, 0, 23.233, 75.018]
  MoveL 1715 to (8.05, 34, -2.75) mm, rotated rx -180 ry 0 rz 90 deg; joints [74.991, -17.759, 84.675, 0, 23.084, 74.991]
  MoveC 1716 to (6.12, 33.77, -2.75) mm, rotated rx -180 ry 0 rz 90 deg; joints [74.967, -17.793, 84.808, 0, 22.986, 74.967] to (4.26, 33.21, -2.75) mm, rotated rx 180 ry 0 rz 90 deg; joints [74.932, -17.825, 84.929, 0, 22.896, 74.932]
  MoveC 1717 to (1.32, 30.73, -2.75) mm, rotated rx 180 ry 0 rz 90 deg; joints [74.825, -17.866, 85.09, 0, 22.776, 74.825] to (0.38, 27, -2.75) mm, rotated rx 180 ry 0 rz 90 deg; joints [74.695, -17.865, 85.085, 0, 22.78, 74.695]
  MoveC 1718 to (0.58, 25.53, -2.75) mm, rotated rx -180 ry 0 rz 90 deg; joints [74.649, -17.854, 85.042, 0, 22.812, 74.649] to (0.99, 24.1, -2.75) mm, rotated rx -180 ry 0 rz 90 deg; joints [74.606, -17.839, 84.985, 0, 22.854, 74.606]
  MoveL 1719 to (6.46, 9, -2.75) mm, rotated rx 180 ry 0 rz 90 deg; joints [74.166, -17.66, 84.297, 0, 23.363, 74.166]
  MoveL 1720 to (7.05, 7.41, -2.75) mm, rotated rx -180 ry 0 rz 90 deg; joints [74.12, -17.641, 84.223, 0, 23.418, 74.12]
  MoveC 1721 to (8.04, 5.58, -2.75) mm, rotated rx 180 ry 0 rz 90 deg; joints [74.07, -17.613, 84.115, 0, 23.497, 74.07] to (9.49, 4.08, -2.75) mm, rotated rx 180 ry 0 rz 90 deg; joints [74.035, -17.577, 83.982, 0, 23.596, 74.035]
  MoveL 1722 to (26.06, -8.81, -2.75) mm, rotated rx -180 ry 0 rz 90 deg; joints [73.776, -17.186, 82.522, 0, 24.664, 73.776]
  MoveL 1723 to (26.96, -9.48, -2.75) mm, rotated rx 180 ry 0 rz 90 deg; joints [73.762, -17.164, 82.442, 0, 24.722, 73.762]
  MoveC 1724 to (31.96, -10.8, -2.75) mm, rotated rx 180 ry 0 rz 90 deg; joints [73.767, -17.056, 82.051, 0, 25.005, 73.767] to (36.45, -8.24, -2.75) mm, rotated rx -180 ry 0 rz 90 deg; joints [73.889, -16.981, 81.778, 0, 25.203, 73.889]
  MoveL 1725 to (37.34, -7.11, -2.75) mm, rotated rx 180 ry 0 rz 90 deg; joints [73.933, -16.969, 81.737, 0, 25.233, 73.933]
  MoveL 1726 to (59.75, 24.17, -2.75) mm, rotated rx -180 ry 0 rz 90 deg; joints [75.118, -16.685, 80.721, 0, 25.964, 75.118]
  MoveC 1727 to (60.59, 25.52, -2.75) mm, rotated rx 180 ry 0 rz 90 deg; joints [75.168, -16.675, 80.685, 0, 25.989, 75.168] to (61.23, 26.97, -2.75) mm, rotated rx 180 ry 0 rz 90 deg; joints [75.219, -16.669, 80.666, 0, 26.003, 75.219]
  MoveC 1728 to (60.51, 32.49, -2.75) mm, rotated rx 180 ry 0 rz 90 deg; joints [75.387, -16.715, 80.828, 0, 25.887, 75.387] to (55.64, 35.18, -2.75) mm, rotated rx -180 ry 0 rz 90 deg; joints [75.433, -16.831, 81.241, 0, 25.59, 75.433]
  MoveL 1729 to (54.49, 35.22, -2.75) mm, rotated rx -180 ry 0 rz 90 deg; joints [75.425, -16.855, 81.327, 0, 25.528, 75.425]
  MoveL 1730 to (45.01, 35, -2.75) mm, rotated rx 180 ry 0 rz 90 deg; joints [75.339, -17.048, 82.022, 0, 25.027, 75.339]
  MoveL 1731 to (41.22, 34.89, -2.75) mm, rotated rx 180 ry 0 rz 90 deg; joints [75.304, -17.124, 82.298, 0, 24.827, 75.304]
  MoveL 1732 to (31.85, 34.64, -2.75) mm, rotated rx 180 ry 0 rz 90 deg; joints [75.216, -17.309, 82.976, 0, 24.333, 75.216]
  MoveL 1733 to (32.05, 27.09, -2.75) mm, rotated rx 180 ry 0 rz 90 deg; joints [74.976, -17.265, 82.815, 0, 24.45, 74.976]
  MoveL 1734 to (32.05, 27.09, 0.25) mm, rotated rx 180 ry 0 rz 90 deg; joints [74.976, -17.418, 82.916, 0, 24.501, 74.976]
  Establecer velocidad (1000.0 mm/s)
  MoveL 1735 to (32.05, 27.09, 10) mm, rotated rx 180 ry 0 rz 90 deg; joints [74.976, -17.912, 83.241, 0, 24.671, 74.976]
  Establecer velocidad (66.7 mm/s)
  MoveL 1736 to (69.27, -30.26, 10) mm, rotated rx 180 ry 0 rz 90 deg; joints [73.501, -16.787, 79.291, 0, 27.496, 73.501]
  MoveL 1737 to (69.27, -30.26, 0.5) mm, rotated rx 180 ry 0 rz 90 deg; joints [73.501, -16.312, 78.972, 0, 27.339, 73.501]
  MoveL 1738 to (70.78, -30.45, 0.09) mm, rotated rx 180 ry 0 rz 90 deg; joints [73.509, -16.257, 78.841, 0, 27.416, 73.509]
  MoveL 1739 to (72.29, -30.26, -0.31) mm, rotated rx -180 ry 0 rz 90 deg; joints [73.528, -16.204, 78.717, 0, 27.487, 73.528]
  MoveL 1740 to (73.72, -29.75, -0.72) mm, rotated rx 180 ry 0 rz 90 deg; joints [73.557, -16.155, 78.606, 0, 27.549, 73.557]
  MoveL 1741 to (75, -28.94, -1.13) mm, rotated rx 180 ry 0 rz 90 deg; joints [73.594, -16.112, 78.514, 0, 27.598, 73.594]
  MoveL 1742 to (76.07, -27.86, -1.53) mm, rotated rx 180 ry 0 rz 90 deg; joints [73.637, -16.074, 78.443, 0, 27.631, 73.637]
  MoveL 1743 to (76.87, -26.57, -1.94) mm, rotated rx 180 ry 0 rz 90 deg; joints [73.684, -16.044, 78.397, 0, 27.648, 73.684]
  MoveL 1744 to (77.37, -25.13, -2.34) mm, rotated rx 180 ry 0 rz 90 deg; joints [73.733, -16.022, 78.377, 0, 27.645, 73.733]
  MoveL 1745 to (77.51, -23.62, -2.75) mm, rotated rx 180 ry 0 rz 90 deg; joints [73.78, -16.009, 78.386, 0, 27.623, 73.78]
  MoveL 1746 to (77.51, -5.21, -2.75) mm, rotated rx 180 ry 0 rz 90 deg; joints [74.35, -16.126, 78.785, 0, 27.341, 74.35]
  MoveC 1747 to (77.45, -3.24, -2.75) mm, rotated rx 180 ry 0 rz 90 deg; joints [74.411, -16.14, 78.831, 0, 27.309, 74.411] to (77.23, -1.29, -2.75) mm, rotated rx -180 ry 0 rz 90 deg; joints [74.47, -16.157, 78.889, 0, 27.268, 74.47]
  MoveC 1748 to (73.65, 2.77, -2.75) mm, rotated rx 180 ry 0 rz 90 deg; joints [74.565, -16.261, 79.245, 0, 27.016, 74.565] to (68.23, 2.92, -2.75) mm, rotated rx 180 ry 0 rz 90 deg; joints [74.523, -16.38, 79.656, 0, 26.724, 74.523]
  MoveL 1749 to (67.76, 2.56, -2.75) mm, rotated rx -180 ry 0 rz 90 deg; joints [74.508, -16.388, 79.684, 0, 26.704, 74.508]
  MoveL 1750 to (65.91, 0.47, -2.75) mm, rotated rx 180 ry 0 rz 90 deg; joints [74.426, -16.416, 79.78, 0, 26.636, 74.426]
  MoveL 1751 to (65.2, -0.47, -2.75) mm, rotated rx 180 ry 0 rz 90 deg; joints [74.39, -16.425, 79.813, 0, 26.613, 74.39]
  MoveL 1752 to (49.31, -22.27, -2.75) mm, rotated rx 180 ry 0 rz 90 deg; joints [73.566, -16.631, 80.53, 0, 26.101, 73.566]
  MoveC 1753 to (48.11, -26.39, -2.75) mm, rotated rx -180 ry 0 rz 90 deg; joints [73.426, -16.63, 80.529, 0, 26.101, 73.426] to (49.75, -30.35, -2.75) mm, rotated rx 180 ry 0 rz 90 deg; joints [73.317, -16.571, 80.319, 0, 26.251, 73.317]
  MoveL 1754 to (66.08, -48.8, -2.75) mm, rotated rx -180 ry 0 rz 90 deg; joints [72.899, -16.096, 78.681, 0, 27.415, 72.899]
  MoveL 1755 to (66.81, -49.58, -2.75) mm, rotated rx -180 ry 0 rz 90 deg; joints [72.882, -16.074, 78.608, 0, 27.467, 72.882]
  MoveL 1756 to (67.46, -50.21, -2.75) mm, rotated rx 180 ry 0 rz 90 deg; joints [72.869, -16.055, 78.544, 0, 27.512, 72.869]
  MoveC 1757 to (69.51, -51.39, -2.75) mm, rotated rx -180 ry 0 rz 90 deg; joints [72.852, -16.002, 78.362, 0, 27.64, 72.852] to (71.87, -51.46, -2.75) mm, rotated rx 180 ry 0 rz 90 deg; joints [72.872, -15.948, 78.182, 0, 27.767, 72.872]
  MoveL 1758 to (72.42, -51.33, -2.75) mm, rotated rx 180 ry 0 rz 90 deg; joints [72.881, -15.937, 78.143, 0, 27.794, 72.881]
  MoveC 1759 to (75.71, -49.42, -2.75) mm, rotated rx 180 ry 0 rz 90 deg; joints [72.971, -15.875, 77.937, 0, 27.938, 72.971] to (77.34, -45.96, -2.75) mm, rotated rx 180 ry 0 rz 90 deg; joints [73.092, -15.863, 77.894, 0, 27.969, 73.092]
  MoveC 1760 to (77.48, -44.54, -2.75) mm, rotated rx 180 ry 0 rz 90 deg; joints [73.137, -15.869, 77.916, 0, 27.953, 73.137] to (77.51, -43.12, -2.75) mm, rotated rx -180 ry 0 rz 90 deg; joints [73.181, -15.878, 77.946, 0, 27.932, 73.181]
  MoveL 1761 to (77.51, -23.62, -2.75) mm, rotated rx 180 ry 0 rz 90 deg; joints [73.78, -16.009, 78.386, 0, 27.623, 73.78]
  MoveL 1762 to (69.96, -23.62, -2.75) mm, rotated rx 180 ry 0 rz 90 deg; joints [73.712, -16.177, 78.957, 0, 27.219, 73.712]
  MoveL 1763 to (69.96, -23.62, 0.25) mm, rotated rx 180 ry 0 rz 90 deg; joints [73.712, -16.327, 79.059, 0, 27.268, 73.712]
  Establecer velocidad (1000.0 mm/s)
  MoveL 1764 to (69.96, -23.62, 10) mm, rotated rx -180 ry 0 rz 90 deg; joints [73.712, -16.815, 79.387, 0, 27.429, 73.712]
  Establecer velocidad (66.7 mm/s)
  MoveL 1765 to (19.34, -70.8, 10) mm, rotated rx -180 ry 0 rz 90 deg; joints [71.755, -17.58, 82.042, 0, 25.538, 71.755]
  MoveL 1766 to (19.34, -70.8, 0.5) mm, rotated rx 180 ry 0 rz 90 deg; joints [71.755, -17.1, 81.725, 0, 25.375, 71.755]
  MoveL 1767 to (19.17, -72.3, 0.09) mm, rotated rx -180 ry 0 rz 90 deg; joints [71.706, -17.073, 81.688, 0, 25.385, 71.706]
  MoveL 1768 to (19.37, -73.81, -0.31) mm, rotated rx -180 ry 0 rz 90 deg; joints [71.661, -17.038, 81.623, 0, 25.415, 71.661]
  MoveL 1769 to (19.89, -75.23, -0.72) mm, rotated rx 180 ry 0 rz 90 deg; joints [71.622, -16.998, 81.537, 0, 25.46, 71.622]
  MoveL 1770 to (20.72, -76.51, -1.13) mm, rotated rx -180 ry 0 rz 90 deg; joints [71.591, -16.952, 81.433, 0, 25.519, 71.591]
  MoveL 1771 to (21.81, -77.57, -1.53) mm, rotated rx 180 ry 0 rz 90 deg; joints [71.569, -16.902, 81.315, 0, 25.587, 71.569]
  MoveL 1772 to (23.11, -78.36, -1.94) mm, rotated rx 180 ry 0 rz 90 deg; joints [71.558, -16.85, 81.187, 0, 25.662, 71.558]
  MoveL 1773 to (24.55, -78.84, -2.34) mm, rotated rx -180 ry 0 rz 90 deg; joints [71.558, -16.796, 81.057, 0, 25.739, 71.558]
  MoveL 1774 to (26.06, -78.97, -2.75) mm, rotated rx -180 ry 0 rz 90 deg; joints [71.57, -16.744, 80.93, 0, 25.814, 71.57]
  MoveL 1775 to (52.59, -78.7, -2.75) mm, rotated rx 180 ry 0 rz 90 deg; joints [71.849, -16.183, 78.98, 0, 27.204, 71.849]
  MoveL 1776 to (54.49, -78.62, -2.75) mm, rotated rx -180 ry 0 rz 90 deg; joints [71.87, -16.142, 78.84, 0, 27.303, 71.87]
  MoveC 1777 to (56.59, -78.23, -2.75) mm, rotated rx -180 ry 0 rz 90 deg; joints [71.903, -16.099, 78.692, 0, 27.407, 71.903] to (58.48, -77.23, -2.75) mm, rotated rx 180 ry 0 rz 90 deg; joints [71.953, -16.065, 78.575, 0, 27.49, 71.953]
  MoveC 1778 to (60.71, -73.02, -2.75) mm, rotated rx 180 ry 0 rz 90 deg; joints [72.104, -16.045, 78.51, 0, 27.535, 72.104] to (59.42, -68.43, -2.75) mm, rotated rx 180 ry 0 rz 90 deg; joints [72.232, -16.107, 78.718, 0, 27.389, 72.232]
  MoveL 1779 to (58.28, -66.94, -2.75) mm, rotated rx -180 ry 0 rz 90 deg; joints [72.266, -16.142, 78.839, 0, 27.303, 72.266]
  MoveL 1780 to (51.64, -59.23, -2.75) mm, rotated rx 180 ry 0 rz 90 deg; joints [72.439, -16.34, 79.519, 0, 26.822, 72.439]
  MoveL 1781 to (50.82, -58.28, -2.75) mm, rotated rx 180 ry 0 rz 90 deg; joints [72.46, -16.364, 79.601, 0, 26.763, 72.46]
  MoveL 1782 to (29.85, -34.02, -2.75) mm, rotated rx 180 ry 0 rz 90 deg; joints [73.013, -16.959, 81.7, 0, 25.259, 73.013]
  MoveL 1783 to (28.75, -32.81, -2.75) mm, rotated rx 180 ry 0 rz 90 deg; joints [73.041, -16.989, 81.807, 0, 25.182, 73.041]
  MoveL 1784 to (27.96, -32.15, -2.75) mm, rotated rx 180 ry 0 rz 90 deg; joints [73.054, -17.009, 81.879, 0, 25.13, 73.054]
  MoveL 1785 to (13.96, -20.98, -2.75) mm, rotated rx -180 ry 0 rz 90 deg; joints [73.274, -17.352, 83.135, 0, 24.217, 73.274]
  MoveC 1786 to (12.21, -19.83, -2.75) mm, rotated rx 180 ry 0 rz 90 deg; joints [73.294, -17.392, 83.285, 0, 24.107, 73.294] to (10.27, -19.04, -2.75) mm, rotated rx 180 ry 0 rz 90 deg; joints [73.301, -17.434, 83.441, 0, 23.993, 73.301]
  MoveC 1787 to (5.61, -19.4, -2.75) mm, rotated rx -180 ry 0 rz 90 deg; joints [73.244, -17.52, 83.766, 0, 23.754, 73.244] to (2.45, -22.85, -2.75) mm, rotated rx 180 ry 0 rz 90 deg; joints [73.103, -17.56, 83.917, 0, 23.643, 73.103]
  MoveL 1788 to (1.94, -24.17, -2.75) mm, rotated rx 180 ry 0 rz 90 deg; joints [73.056, -17.562, 83.925, 0, 23.638, 73.056]
  MoveL 1789 to (0.47, -29.65, -2.75) mm, rotated rx -180 ry 0 rz 90 deg; joints [72.866, -17.558, 83.909, 0, 23.649, 72.866]
  MoveL 1790 to (-10.16, -69.65, -2.75) mm, rotated rx -180 ry 0 rz 90 deg; joints [71.483, -17.517, 83.752, 0, 23.765, 71.483]
  MoveL 1791 to (-10.38, -70.6, -2.75) mm, rotated rx 180 ry 0 rz 90 deg; joints [71.45, -17.515, 83.744, 0, 23.77, 71.45]
  MoveC 1792 to (-9.54, -75.85, -2.75) mm, rotated rx 180 ry 0 rz 90 deg; joints [71.293, -17.466, 83.56, 0, 23.905, 71.293] to (-5.21, -78.94, -2.75) mm, rotated rx 180 ry 0 rz 90 deg; joints [71.242, -17.364, 83.18, 0, 24.184, 71.242]
  MoveC 1793 to (-3.8, -79.19, -2.75) mm, rotated rx 180 ry 0 rz 90 deg; joints [71.249, -17.335, 83.074, 0, 24.262, 71.249] to (-2.37, -79.26, -2.75) mm, rotated rx 180 ry 0 rz 90 deg; joints [71.262, -17.307, 82.97, 0, 24.337, 71.262]
  MoveL 1794 to (26.06, -78.97, -2.75) mm, rotated rx -180 ry 0 rz 90 deg; joints [71.57, -16.744, 80.93, 0, 25.814, 71.57]
  MoveL 1795 to (25.98, -71.42, -2.75) mm, rotated rx 180 ry 0 rz 90 deg; joints [71.804, -16.797, 81.118, 0, 25.679, 71.804]
  MoveL 1796 to (25.98, -71.42, 0.25) mm, rotated rx -180 ry 0 rz 90 deg; joints [71.804, -16.948, 81.219, 0, 25.729, 71.804]
  Establecer velocidad (1000.0 mm/s)
  MoveL 1797 to (25.98, -71.42, 10) mm, rotated rx -180 ry 0 rz 90 deg; joints [71.804, -17.44, 81.545, 0, 25.895, 71.804]
  Establecer velocidad (66.7 mm/s)
  MoveL 1798 to (-71.71, -45.07, 10) mm, rotated rx -180 ry 0 rz 90 deg; joints [71.613, -19.378, 88.976, 0, 20.402, 71.613]
  MoveL 1799 to (-71.71, -45.07, 0.5) mm, rotated rx -180 ry 0 rz 90 deg; joints [71.613, -18.885, 88.661, 0, 20.224, 71.613]
  MoveL 1800 to (-73.22, -44.88, 0.09) mm, rotated rx 180 ry 0 rz 90 deg; joints [71.603, -18.888, 88.752, 0, 20.136, 71.603]
  MoveL 1801 to (-74.73, -45.07, -0.31) mm, rotated rx 180 ry 0 rz 90 deg; joints [71.58, -18.889, 88.836, 0, 20.054, 71.58]
  MoveL 1802 to (-76.16, -45.58, -0.72) mm, rotated rx 180 ry 0 rz 90 deg; joints [71.548, -18.888, 88.906, 0, 19.982, 71.548]
  MoveL 1803 to (-77.44, -46.4, -1.13) mm, rotated rx 180 ry 0 rz 90 deg; joints [71.506, -18.882, 88.96, 0, 19.922, 71.506]
  MoveL 1804 to (-78.51, -47.48, -1.53) mm, rotated rx -180 ry 0 rz 90 deg; joints [71.459, -18.872, 88.994, 0, 19.878, 71.459]
  MoveL 1805 to (-79.31, -48.77, -1.94) mm, rotated rx 180 ry 0 rz 90 deg; joints [71.407, -18.856, 89.005, 0, 19.852, 71.407]
  MoveL 1806 to (-79.81, -50.2, -2.34) mm, rotated rx -180 ry 0 rz 90 deg; joints [71.354, -18.836, 88.992, 0, 19.843, 71.354]
  MoveL 1807 to (-79.95, -51.71, -2.75) mm, rotated rx -180 ry 0 rz 90 deg; joints [71.303, -18.809, 88.954, 0, 19.855, 71.303]
  MoveL 1808 to (-79.95, -71.06, -2.75) mm, rotated rx 180 ry 0 rz 90 deg; joints [70.665, -18.705, 88.509, 0, 20.197, 70.665]
  MoveC 1809 to (-78.17, -76.16, -2.75) mm, rotated rx 180 ry 0 rz 90 deg; joints [70.519, -18.649, 88.27, 0, 20.38, 70.519] to (-73.6, -79.04, -2.75) mm, rotated rx 180 ry 0 rz 90 deg; joints [70.478, -18.561, 87.895, 0, 20.665, 70.478]
  MoveC 1810 to (-72.27, -79.26, -2.75) mm, rotated rx -180 ry 0 rz 90 deg; joints [70.486, -18.538, 87.801, 0, 20.738, 70.486] to (-70.92, -79.33, -2.75) mm, rotated rx 180 ry 0 rz 90 deg; joints [70.499, -18.516, 87.708, 0, 20.808, 70.499]
  MoveL 1811 to (-35.26, -79.03, -2.75) mm, rotated rx -180 ry 0 rz 90 deg; joints [70.912, -17.916, 85.283, 0, 22.633, 70.912]
  MoveC 1812 to (-30.12, -77.24, -2.75) mm, rotated rx -180 ry 0 rz 90 deg; joints [71.026, -17.835, 84.969, 0, 22.866, 71.026] to (-27.13, -72.69, -2.75) mm, rotated rx 180 ry 0 rz 90 deg; joints [71.204, -17.809, 84.87, 0, 22.94, 71.204]
  MoveL 1813 to (-14.49, -24.17, -2.75) mm, rotated rx 180 ry 0 rz 90 deg; joints [72.894, -17.865, 85.085, 0, 22.78, 72.894]
  MoveC 1814 to (-14.21, -20.27, -2.75) mm, rotated rx 180 ry 0 rz 90 deg; joints [73.023, -17.881, 85.149, 0, 22.732, 73.023] to (-15.53, -16.58, -2.75) mm, rotated rx 180 ry 0 rz 90 deg; joints [73.129, -17.925, 85.32, 0, 22.605, 73.129]
  MoveC 1815 to (-18.94, -13.96, -2.75) mm, rotated rx 180 ry 0 rz 90 deg; joints [73.181, -18, 85.614, 0, 22.386, 73.181] to (-23.22, -13.54, -2.75) mm, rotated rx 180 ry 0 rz 90 deg; joints [73.152, -18.078, 85.921, 0, 22.156, 73.152]
  MoveL 1816 to (-25.11, -13.9, -2.75) mm, rotated rx -180 ry 0 rz 90 deg; joints [73.122, -18.109, 86.046, 0, 22.063, 73.122]
  MoveL 1817 to (-72.49, -23.97, -2.75) mm, rotated rx 180 ry 0 rz 90 deg; joints [72.305, -18.834, 89.065, 0, 19.769, 72.305]
  MoveL 1818 to (-73.48, -24.2, -2.75) mm, rotated rx -180 ry 0 rz 90 deg; joints [72.286, -18.848, 89.126, 0, 19.722, 72.286]
  MoveC 1819 to (-78.14, -27.16, -2.75) mm, rotated rx 180 ry 0 rz 90 deg; joints [72.138, -18.905, 89.374, 0, 19.531, 72.138] to (-79.95, -32.36, -2.75) mm, rotated rx 180 ry 0 rz 90 deg; joints [71.945, -18.907, 89.382, 0, 19.524, 71.945]
  MoveL 1820 to (-79.95, -51.71, -2.75) mm, rotated rx -180 ry 0 rz 90 deg; joints [71.303, -18.809, 88.954, 0, 19.855, 71.303]
  MoveL 1821 to (-72.4, -51.71, -2.75) mm, rotated rx -180 ry 0 rz 90 deg; joints [71.387, -18.691, 88.449, 0, 20.243, 71.387]
  MoveL 1822 to (-72.4, -51.71, 0.25) mm, rotated rx -180 ry 0 rz 90 deg; joints [71.387, -18.847, 88.55, 0, 20.298, 71.387]
  Establecer velocidad (1000.0 mm/s)
  MoveL 1823 to (-72.4, -51.71, 10) mm, rotated rx -180 ry 0 rz 90 deg; joints [71.387, -19.354, 88.874, 0, 20.481, 71.387]
  Establecer velocidad (66.7 mm/s)
  MoveL 1824 to (-71.71, 36.34, 10) mm, rotated rx 180 ry 0 rz 90 deg; joints [74.341, -19.763, 90.648, 0, 19.115, 74.341]
  MoveL 1825 to (-71.71, 36.34, 0.5) mm, rotated rx 180 ry 0 rz 90 deg; joints [74.341, -19.265, 90.332, 0, 18.933, 74.341]
  MoveL 1826 to (-73.22, 36.52, 0.09) mm, rotated rx 180 ry 0 rz 90 deg; joints [74.333, -19.267, 90.422, 0, 18.845, 74.333]
  MoveL 1827 to (-74.72, 36.34, -0.31) mm, rotated rx 180 ry 0 rz 90 deg; joints [74.313, -19.267, 90.506, 0, 18.761, 74.313]
  MoveL 1828 to (-76.16, 35.83, -0.72) mm, rotated rx -180 ry 0 rz 90 deg; joints [74.282, -19.264, 90.578, 0, 18.686, 74.282]
  MoveL 1829 to (-77.44, 35.01, -1.13) mm, rotated rx 180 ry 0 rz 90 deg; joints [74.242, -19.258, 90.635, 0, 18.624, 74.242]
  MoveL 1830 to (-78.51, 33.93, -1.53) mm, rotated rx -180 ry 0 rz 90 deg; joints [74.194, -19.248, 90.672, 0, 18.576, 74.194]
  MoveL 1831 to (-79.31, 32.64, -1.94) mm, rotated rx 180 ry 0 rz 90 deg; joints [74.143, -19.233, 90.687, 0, 18.546, 74.143]
  MoveL 1832 to (-79.81, 31.21, -2.34) mm, rotated rx -180 ry 0 rz 90 deg; joints [74.089, -19.213, 90.68, 0, 18.533, 74.089]
  MoveL 1833 to (-79.95, 29.7, -2.75) mm, rotated rx -180 ry 0 rz 90 deg; joints [74.036, -19.188, 90.647, 0, 18.541, 74.036]
  MoveL 1834 to (-79.95, 0.47, -2.75) mm, rotated rx -180 ry 0 rz 90 deg; joints [73.046, -19.061, 90.072, 0, 18.989, 73.046]
  MoveC 1835 to (-77.15, -5.76, -2.75) mm, rotated rx -180 ry 0 rz 90 deg; joints [72.864, -18.991, 89.758, 0, 19.233, 72.864] to (-70.6, -7.71, -2.75) mm, rotated rx 180 ry 0 rz 90 deg; joints [72.867, -18.883, 89.28, 0, 19.604, 72.867]
  MoveL 1836 to (-69.65, -7.57, -2.75) mm, rotated rx 180 ry 0 rz 90 deg; joints [72.881, -18.869, 89.219, 0, 19.65, 72.881]
  MoveL 1837 to (-63.97, -6.28, -2.75) mm, rotated rx -180 ry 0 rz 90 deg; joints [72.983, -18.788, 88.863, 0, 19.924, 72.983]
  MoveL 1838 to (-63.02, -6.06, -2.75) mm, rotated rx -180 ry 0 rz 90 deg; joints [73, -18.774, 88.804, 0, 19.97, 73]
  MoveL 1839 to (-23.22, 3.09, -2.75) mm, rotated rx 180 ry 0 rz 90 deg; joints [73.696, -18.164, 86.266, 0, 21.898, 73.696]
  MoveL 1840 to (-19.52, 3.95, -2.75) mm, rotated rx -180 ry 0 rz 90 deg; joints [73.759, -18.104, 86.026, 0, 22.078, 73.759]
  MoveC 1841 to (-14.25, 7.91, -2.75) mm, rotated rx 180 ry 0 rz 90 deg; joints [73.938, -18.031, 85.738, 0, 22.293, 73.938] to (-13.62, 14.47, -2.75) mm, rotated rx 180 ry 0 rz 90 deg; joints [74.159, -18.053, 85.825, 0, 22.228, 74.159]
  MoveL 1842 to (-14.01, 15.64, -2.75) mm, rotated rx 180 ry 0 rz 90 deg; joints [74.193, -18.066, 85.875, 0, 22.191, 74.193]
  MoveL 1843 to (-20.59, 33.99, -2.75) mm, rotated rx -180 ry 0 rz 90 deg; joints [74.737, -18.269, 86.69, 0, 21.579, 74.737]
  MoveC 1844 to (-21.89, 36.36, -2.75) mm, rotated rx 180 ry 0 rz 90 deg; joints [74.803, -18.302, 86.826, 0, 21.476, 74.803] to (-23.88, 38.2, -2.75) mm, rotated rx -180 ry 0 rz 90 deg; joints [74.846, -18.345, 86.999, 0, 21.346, 74.846]
  MoveL 1845 to (-25.11, 39.03, -2.75) mm, rotated rx 180 ry 0 rz 90 deg; joints [74.863, -18.369, 87.1, 0, 21.27, 74.863]
  MoveL 1846 to (-66.34, 65.47, -2.75) mm, rotated rx 180 ry 0 rz 90 deg; joints [75.384, -19.132, 90.391, 0, 18.741, 75.384]
  MoveC 1847 to (-68.83, 66.7, -2.75) mm, rotated rx 180 ry 0 rz 90 deg; joints [75.404, -19.173, 90.579, 0, 18.594, 75.404] to (-71.52, 67.34, -2.75) mm, rotated rx -180 ry 0 rz 90 deg; joints [75.402, -19.214, 90.771, 0, 18.444, 75.402]
  MoveC 1848 to (-76.03, 66.44, -2.75) mm, rotated rx 180 ry 0 rz 90 deg; joints [75.331, -19.276, 91.055, 0, 18.22, 75.331] to (-79.1, 63.02, -2.75) mm, rotated rx -180 ry 0 rz 90 deg; joints [75.185, -19.307, 91.2, 0, 18.107, 75.185]
  MoveC 1849 to (-79.74, 61.01, -2.75) mm, rotated rx 180 ry 0 rz 90 deg; joints [75.11, -19.308, 91.207, 0, 18.101, 75.11] to (-79.95, 58.92, -2.75) mm, rotated rx -180 ry 0 rz 90 deg; joints [75.036, -19.303, 91.184, 0, 18.119, 75.036]
  MoveL 1850 to (-79.95, 29.7, -2.75) mm, rotated rx -180 ry 0 rz 90 deg; joints [74.036, -19.188, 90.647, 0, 18.541, 74.036]
  MoveL 1851 to (-72.4, 29.7, -2.75) mm, rotated rx 180 ry 0 rz 90 deg; joints [74.109, -19.077, 90.143, 0, 18.934, 74.109]
  MoveL 1852 to (-72.4, 29.7, 0.25) mm, rotated rx 180 ry 0 rz 90 deg; joints [74.109, -19.234, 90.244, 0, 18.991, 74.109]
  Establecer velocidad (1000.0 mm/s)
  MoveL 1853 to (-72.4, 29.7, 10) mm, rotated rx 180 ry 0 rz 90 deg; joints [74.109, -19.745, 90.568, 0, 19.177, 74.109]
  Establecer velocidad (66.7 mm/s)
  MoveL 1854 to (-71.34, 36.34, 10) mm, rotated rx 180 ry 0 rz 90 deg; joints [74.345, -19.757, 90.623, 0, 19.135, 74.345]
  MoveL 1855 to (-71.34, 36.34, 0.25) mm, rotated rx -180 ry 0 rz 90 deg; joints [74.345, -19.246, 90.298, 0, 18.948, 74.345]
  MoveL 1856 to (-72.85, 36.52, -0.16) mm, rotated rx 180 ry 0 rz 90 deg; joints [74.337, -19.248, 90.389, 0, 18.859, 74.337]
  MoveL 1857 to (-74.35, 36.34, -0.56) mm, rotated rx 180 ry 0 rz 90 deg; joints [74.316, -19.248, 90.473, 0, 18.776, 74.316]
  MoveL 1858 to (-75.79, 35.83, -0.97) mm, rotated rx -180 ry 0 rz 90 deg; joints [74.285, -19.246, 90.545, 0, 18.701, 74.285]
  MoveL 1859 to (-77.07, 35.01, -1.37) mm, rotated rx -180 ry 0 rz 90 deg; joints [74.245, -19.24, 90.602, 0, 18.638, 74.245]
  MoveL 1860 to (-78.14, 33.93, -1.78) mm, rotated rx -180 ry 0 rz 90 deg; joints [74.198, -19.23, 90.639, 0, 18.591, 74.198]
  MoveL 1861 to (-78.94, 32.64, -2.19) mm, rotated rx 180 ry 0 rz 90 deg; joints [74.146, -19.215, 90.654, 0, 18.56, 74.146]
  MoveL 1862 to (-79.44, 31.21, -2.59) mm, rotated rx -180 ry 0 rz 90 deg; joints [74.092, -19.195, 90.647, 0, 18.548, 74.092]
  MoveL 1863 to (-79.58, 29.7, -3) mm, rotated rx 180 ry 0 rz 90 deg; joints [74.04, -19.169, 90.614, 0, 18.556, 74.04]
  MoveL 1864 to (-79.58, 0.47, -3) mm, rotated rx 180 ry 0 rz 90 deg; joints [73.049, -19.043, 90.039, 0, 19.004, 73.049]
  MoveC 1865 to (-78.72, -3.17, -3) mm, rotated rx -180 ry 0 rz 90 deg; joints [72.936, -19.014, 89.907, 0, 19.106, 72.936] to (-76.29, -6.02, -3) mm, rotated rx 180 ry 0 rz 90 deg; joints [72.865, -18.964, 89.687, 0, 19.278, 72.865]
  MoveC 1866 to (-72.94, -7.27, -3) mm, rotated rx -180 ry 0 rz 90 deg; joints [72.858, -18.908, 89.437, 0, 19.471, 72.858] to (-69.37, -7.11, -3) mm, rotated rx 180 ry 0 rz 90 deg; joints [72.9, -18.854, 89.201, 0, 19.653, 72.9]
  MoveL 1867 to (-19.61, 4.34, -3) mm, rotated rx 180 ry 0 rz 90 deg; joints [73.771, -18.094, 86.031, 0, 22.063, 73.771]
  MoveC 1868 to (-14.73, 7.86, -3) mm, rotated rx -180 ry 0 rz 90 deg; joints [73.932, -18.027, 85.762, 0, 22.265, 73.932] to (-13.86, 13.8, -3) mm, rotated rx 180 ry 0 rz 90 deg; joints [74.135, -18.041, 85.82, 0, 22.222, 74.135]
  MoveL 1869 to (-14.08, 14.69, -3) mm, rotated rx 180 ry 0 rz 90 deg; joints [74.161, -18.05, 85.853, 0, 22.196, 74.161]
  MoveL 1870 to (-15.64, 19.03, -3) mm, rotated rx -180 ry 0 rz 90 deg; joints [74.289, -18.099, 86.048, 0, 22.051, 74.289]
  MoveL 1871 to (-20.89, 33.75, -3) mm, rotated rx -180 ry 0 rz 90 deg; joints [74.726, -18.26, 86.699, 0, 21.561, 74.726]
  MoveC 1872 to (-22.24, 36.18, -3) mm, rotated rx 180 ry 0 rz 90 deg; joints [74.794, -18.295, 86.839, 0, 21.456, 74.794] to (-24.31, 38.04, -3) mm, rotated rx 180 ry 0 rz 90 deg; joints [74.837, -18.338, 87.017, 0, 21.321, 74.837]
  MoveL 1873 to (-66.81, 65.31, -3) mm, rotated rx -180 ry 0 rz 90 deg; joints [75.375, -19.125, 90.411, 0, 18.714, 75.375]
  MoveC 1874 to (-69.17, 66.41, -3) mm, rotated rx 180 ry 0 rz 90 deg; joints [75.391, -19.164, 90.589, 0, 18.575, 75.391] to (-71.72, 66.97, -3) mm, rotated rx 180 ry 0 rz 90 deg; joints [75.388, -19.203, 90.769, 0, 18.434, 75.388]
  MoveC 1875 to (-76.03, 65.99, -3) mm, rotated rx -180 ry 0 rz 90 deg; joints [75.316, -19.261, 91.039, 0, 18.222, 75.316] to (-78.85, 62.61, -3) mm, rotated rx -180 ry 0 rz 90 deg; joints [75.173, -19.288, 91.168, 0, 18.12, 75.173]
  MoveC 1876 to (-79.4, 60.69, -3) mm, rotated rx 180 ry 0 rz 90 deg; joints [75.102, -19.289, 91.17, 0, 18.119, 75.102] to (-79.58, 58.7, -3) mm, rotated rx 180 ry 0 rz 90 deg; joints [75.032, -19.284, 91.147, 0, 18.137, 75.032]
  MoveL 1877 to (-79.58, 29.7, -3) mm, rotated rx 180 ry 0 rz 90 deg; joints [74.04, -19.169, 90.614, 0, 18.556, 74.04]
  MoveL 1878 to (-72.03, 29.7, -3) mm, rotated rx -180 ry 0 rz 90 deg; joints [74.113, -19.059, 90.11, 0, 18.949, 74.113]
  MoveL 1879 to (-72.03, 29.7, 0) mm, rotated rx 180 ry 0 rz 90 deg; joints [74.113, -19.216, 90.211, 0, 19.005, 74.113]
  Establecer velocidad (1000.0 mm/s)
  MoveL 1880 to (-72.03, 29.7, 10) mm, rotated rx -180 ry 0 rz 90 deg; joints [74.113, -19.74, 90.543, 0, 19.196, 74.113]
  Establecer velocidad (66.7 mm/s)
  MoveL 1881 to (-71.34, -45.04, 10) mm, rotated rx 180 ry 0 rz 90 deg; joints [71.618, -19.373, 88.952, 0, 20.421, 71.618]
  MoveL 1882 to (-71.34, -45.04, 0.25) mm, rotated rx -180 ry 0 rz 90 deg; joints [71.618, -18.866, 88.628, 0, 20.238, 71.618]
  MoveL 1883 to (-72.85, -44.86, -0.16) mm, rotated rx -180 ry 0 rz 90 deg; joints [71.608, -18.869, 88.72, 0, 20.15, 71.608]
  MoveL 1884 to (-74.36, -45.04, -0.56) mm, rotated rx -180 ry 0 rz 90 deg; joints [71.585, -18.871, 88.803, 0, 20.068, 71.585]
  MoveL 1885 to (-75.79, -45.55, -0.97) mm, rotated rx -180 ry 0 rz 90 deg; joints [71.553, -18.869, 88.874, 0, 19.996, 71.553]
  MoveL 1886 to (-77.07, -46.37, -1.37) mm, rotated rx 180 ry 0 rz 90 deg; joints [71.511, -18.864, 88.928, 0, 19.936, 71.511]
  MoveL 1887 to (-78.14, -47.45, -1.78) mm, rotated rx -180 ry 0 rz 90 deg; joints [71.464, -18.853, 88.961, 0, 19.892, 71.464]
  MoveL 1888 to (-78.94, -48.74, -2.19) mm, rotated rx 180 ry 0 rz 90 deg; joints [71.412, -18.838, 88.972, 0, 19.866, 71.412]
  MoveL 1889 to (-79.44, -50.18, -2.59) mm, rotated rx 180 ry 0 rz 90 deg; joints [71.359, -18.817, 88.96, 0, 19.857, 71.359]
  MoveL 1890 to (-79.58, -51.68, -3) mm, rotated rx 180 ry 0 rz 90 deg; joints [71.308, -18.79, 88.921, 0, 19.869, 71.308]
  MoveL 1891 to (-79.58, -70.97, -3) mm, rotated rx 180 ry 0 rz 90 deg; joints [70.672, -18.687, 88.478, 0, 20.209, 70.672]
  MoveC 1892 to (-77.27, -76.58, -3) mm, rotated rx 180 ry 0 rz 90 deg; joints [70.515, -18.62, 88.191, 0, 20.429, 70.515] to (-71.69, -78.94, -3) mm, rotated rx -180 ry 0 rz 90 deg; joints [70.503, -18.518, 87.761, 0, 20.757, 70.503]
  MoveL 1893 to (-70.6, -78.95, -3) mm, rotated rx -180 ry 0 rz 90 deg; joints [70.515, -18.5, 87.687, 0, 20.813, 70.515]
  MoveL 1894 to (-36.48, -78.67, -3) mm, rotated rx -180 ry 0 rz 90 deg; joints [70.909, -17.927, 85.368, 0, 22.559, 70.909]
  MoveL 1895 to (-35.3, -78.66, -3) mm, rotated rx 180 ry 0 rz 90 deg; joints [70.923, -17.906, 85.286, 0, 22.62, 70.923]
  MoveC 1896 to (-30.35, -76.92, -3) mm, rotated rx 180 ry 0 rz 90 deg; joints [71.033, -17.828, 84.984, 0, 22.844, 71.033] to (-27.47, -72.54, -3) mm, rotated rx 180 ry 0 rz 90 deg; joints [71.205, -17.804, 84.889, 0, 22.915, 71.205]
  MoveL 1897 to (-14.88, -24.17, -3) mm, rotated rx 180 ry 0 rz 90 deg; joints [72.89, -17.859, 85.104, 0, 22.755, 72.89]
  MoveC 1898 to (-14.55, -21.8, -3) mm, rotated rx -180 ry 0 rz 90 deg; joints [72.97, -17.866, 85.131, 0, 22.735, 72.97] to (-14.75, -19.43, -3) mm, rotated rx 180 ry 0 rz 90 deg; joints [73.045, -17.883, 85.196, 0, 22.686, 73.045]
  MoveC 1899 to (-16.7, -15.8, -3) mm, rotated rx 180 ry 0 rz 90 deg; joints [73.143, -17.937, 85.41, 0, 22.527, 73.143] to (-20.37, -13.96, -3) mm, rotated rx -180 ry 0 rz 90 deg; joints [73.167, -18.013, 85.706, 0, 22.307, 73.167]
  MoveC 1900 to (-22.27, -13.85, -3) mm, rotated rx 180 ry 0 rz 90 deg; joints [73.152, -18.047, 85.841, 0, 22.206, 73.152] to (-24.17, -14.08, -3) mm, rotated rx -180 ry 0 rz 90 deg; joints [73.125, -18.078, 85.968, 0, 22.111, 73.125]
  MoveL 1901 to (-70.6, -23.96, -3) mm, rotated rx 180 ry 0 rz 90 deg; joints [72.325, -18.792, 88.93, 0, 19.862, 72.325]
  MoveL 1902 to (-73.22, -24.52, -3) mm, rotated rx 180 ry 0 rz 90 deg; joints [72.278, -18.83, 89.093, 0, 19.736, 72.278]
  MoveC 1903 to (-77.79, -27.34, -3) mm, rotated rx 180 ry 0 rz 90 deg; joints [72.136, -18.886, 89.339, 0, 19.547, 72.136] to (-79.58, -32.4, -3) mm, rotated rx -180 ry 0 rz 90 deg; joints [71.948, -18.888, 89.348, 0, 19.539, 71.948]
  MoveL 1904 to (-79.58, -51.68, -3) mm, rotated rx 180 ry 0 rz 90 deg; joints [71.308, -18.79, 88.921, 0, 19.869, 71.308]
  MoveL 1905 to (-72.03, -51.68, -3) mm, rotated rx -180 ry 0 rz 90 deg; joints [71.392, -18.673, 88.416, 0, 20.257, 71.392]
  MoveL 1906 to (-72.03, -51.68, 0) mm, rotated rx 180 ry 0 rz 90 deg; joints [71.392, -18.829, 88.517, 0, 20.312, 71.392]
  Establecer velocidad (1000.0 mm/s)
  MoveL 1907 to (-72.03, -51.68, 10) mm, rotated rx 180 ry 0 rz 90 deg; joints [71.392, -19.348, 88.849, 0, 20.499, 71.392]
  Establecer velocidad (66.7 mm/s)
  MoveL 1908 to (19.23, -70.43, 10) mm, rotated rx 180 ry 0 rz 90 deg; joints [71.765, -17.585, 82.059, 0, 25.526, 71.765]
  MoveL 1909 to (19.23, -70.43, 0.25) mm, rotated rx -180 ry 0 rz 90 deg; joints [71.765, -17.092, 81.733, 0, 25.359, 71.765]
  MoveL 1910 to (19.06, -71.94, -0.16) mm, rotated rx -180 ry 0 rz 90 deg; joints [71.716, -17.065, 81.696, 0, 25.369, 71.716]
  MoveL 1911 to (19.25, -73.45, -0.56) mm, rotated rx -180 ry 0 rz 90 deg; joints [71.671, -17.031, 81.632, 0, 25.399, 71.671]
  MoveL 1912 to (19.78, -74.87, -0.97) mm, rotated rx 180 ry 0 rz 90 deg; joints [71.632, -16.99, 81.546, 0, 25.444, 71.632]
  MoveL 1913 to (20.61, -76.15, -1.37) mm, rotated rx 180 ry 0 rz 90 deg; joints [71.601, -16.944, 81.442, 0, 25.502, 71.601]
  MoveL 1914 to (21.7, -77.21, -1.78) mm, rotated rx 180 ry 0 rz 90 deg; joints [71.58, -16.894, 81.323, 0, 25.571, 71.58]
  MoveL 1915 to (22.99, -78, -2.19) mm, rotated rx -180 ry 0 rz 90 deg; joints [71.568, -16.842, 81.196, 0, 25.646, 71.568]
  MoveL 1916 to (24.43, -78.48, -2.59) mm, rotated rx 180 ry 0 rz 90 deg; joints [71.568, -16.789, 81.066, 0, 25.723, 71.568]
  MoveL 1917 to (25.94, -78.61, -3) mm, rotated rx -180 ry 0 rz 90 deg; joints [71.58, -16.736, 80.939, 0, 25.797, 71.58]
  MoveL 1918 to (26.06, -78.61, -3) mm, rotated rx 180 ry 0 rz 90 deg; joints [71.581, -16.734, 80.931, 0, 25.803, 71.581]
  MoveL 1919 to (53.54, -78.29, -3) mm, rotated rx -180 ry 0 rz 90 deg; joints [71.871, -16.153, 78.91, 0, 27.243, 71.871]
  MoveL 1920 to (54.81, -78.21, -3) mm, rotated rx 180 ry 0 rz 90 deg; joints [71.886, -16.126, 78.818, 0, 27.308, 71.886]
  MoveC 1921 to (57.88, -77.05, -3) mm, rotated rx 180 ry 0 rz 90 deg; joints [71.952, -16.067, 78.616, 0, 27.451, 71.952] to (59.79, -74.39, -3) mm, rotated rx 180 ry 0 rz 90 deg; joints [72.053, -16.043, 78.537, 0, 27.506, 72.053]
  MoveC 1922 to (60.21, -71.46, -3) mm, rotated rx -180 ry 0 rz 90 deg; joints [72.147, -16.055, 78.577, 0, 27.478, 72.147] to (59.13, -68.7, -3) mm, rotated rx 180 ry 0 rz 90 deg; joints [72.22, -16.099, 78.725, 0, 27.374, 72.22]
  MoveL 1923 to (58.45, -67.76, -3) mm, rotated rx 180 ry 0 rz 90 deg; joints [72.243, -16.12, 78.798, 0, 27.322, 72.243]
  MoveL 1924 to (55.22, -63.97, -3) mm, rotated rx -180 ry 0 rz 90 deg; joints [72.328, -16.217, 79.131, 0, 27.087, 72.328]
  MoveL 1925 to (29.84, -34.59, -3) mm, rotated rx -180 ry 0 rz 90 deg; joints [72.995, -16.943, 81.679, 0, 25.264, 72.995]
  MoveL 1926 to (28.5, -33.07, -3) mm, rotated rx 180 ry 0 rz 90 deg; joints [73.03, -16.98, 81.811, 0, 25.169, 73.03]
  MoveL 1927 to (13.47, -21.08, -3) mm, rotated rx -180 ry 0 rz 90 deg; joints [73.266, -17.348, 83.16, 0, 24.188, 73.266]
  MoveC 1928 to (10.92, -19.66, -3) mm, rotated rx 180 ry 0 rz 90 deg; joints [73.287, -17.405, 83.373, 0, 24.032, 73.287] to (8.05, -19.14, -3) mm, rotated rx 180 ry 0 rz 90 deg; joints [73.276, -17.463, 83.589, 0, 23.874, 73.276]
  MoveC 1929 to (4.77, -20.39, -3) mm, rotated rx 180 ry 0 rz 90 deg; joints [73.204, -17.518, 83.796, 0, 23.722, 73.204] to (2.69, -23.22, -3) mm, rotated rx -180 ry 0 rz 90 deg; joints [73.094, -17.541, 83.883, 0, 23.658, 73.094]
  MoveL 1930 to (2.36, -24.17, -3) mm, rotated rx -180 ry 0 rz 90 deg; joints [73.06, -17.542, 83.887, 0, 23.655, 73.06]
  MoveL 1931 to (0.47, -31.15, -3) mm, rotated rx 180 ry 0 rz 90 deg; joints [72.818, -17.537, 83.868, 0, 23.669, 72.818]
  MoveL 1932 to (-0.44, -34.59, -3) mm, rotated rx 180 ry 0 rz 90 deg; joints [72.699, -17.534, 83.857, 0, 23.677, 72.699]
  MoveL 1933 to (-9.77, -69.65, -3) mm, rotated rx 180 ry 0 rz 90 deg; joints [71.487, -17.496, 83.715, 0, 23.781, 71.487]
  MoveL 1934 to (-9.95, -70.51, -3) mm, rotated rx -180 ry 0 rz 90 deg; joints [71.458, -17.494, 83.708, 0, 23.786, 71.458]
  MoveL 1935 to (-9.97, -70.6, -3) mm, rotated rx 180 ry 0 rz 90 deg; joints [71.455, -17.494, 83.707, 0, 23.787, 71.455]
  MoveC 1936 to (-9.47, -75.2, -3) mm, rotated rx -180 ry 0 rz 90 deg; joints [71.314, -17.456, 83.562, 0, 23.893, 71.314] to (-6.05, -78.31, -3) mm, rotated rx 180 ry 0 rz 90 deg; joints [71.253, -17.371, 83.246, 0, 24.125, 71.253]
  MoveC 1937 to (-4.51, -78.75, -3) mm, rotated rx -180 ry 0 rz 90 deg; joints [71.255, -17.339, 83.126, 0, 24.213, 71.255] to (-2.92, -78.88, -3) mm, rotated rx -180 ry 0 rz 90 deg; joints [71.268, -17.308, 83.01, 0, 24.298, 71.268]
  MoveL 1938 to (25.94, -78.61, -3) mm, rotated rx -180 ry 0 rz 90 deg; joints [71.58, -16.736, 80.939, 0, 25.797, 71.58]
  MoveL 1939 to (25.87, -71.06, -3) mm, rotated rx -180 ry 0 rz 90 deg; joints [71.814, -16.789, 81.126, 0, 25.663, 71.814]
  MoveL 1940 to (25.87, -71.06, 0) mm, rotated rx 180 ry 0 rz 90 deg; joints [71.814, -16.94, 81.227, 0, 25.713, 71.814]
  Establecer velocidad (1000.0 mm/s)
  MoveL 1941 to (25.87, -71.06, 10) mm, rotated rx 180 ry 0 rz 90 deg; joints [71.814, -17.445, 81.562, 0, 25.883, 71.814]
  Establecer velocidad (66.7 mm/s)
  MoveL 1942 to (68.88, -30.81, 10) mm, rotated rx 180 ry 0 rz 90 deg; joints [73.48, -16.792, 79.308, 0, 27.484, 73.48]
  MoveL 1943 to (68.88, -30.81, 0.25) mm, rotated rx -180 ry 0 rz 90 deg; joints [73.48, -16.304, 78.981, 0, 27.323, 73.48]
  MoveL 1944 to (70.39, -30.99, -0.16) mm, rotated rx 180 ry 0 rz 90 deg; joints [73.488, -16.249, 78.85, 0, 27.4, 73.488]
  MoveL 1945 to (71.89, -30.81, -0.56) mm, rotated rx -180 ry 0 rz 90 deg; joints [73.508, -16.197, 78.726, 0, 27.471, 73.508]
  MoveL 1946 to (73.33, -30.3, -0.97) mm, rotated rx 180 ry 0 rz 90 deg; joints [73.537, -16.148, 78.615, 0, 27.533, 73.537]
  MoveL 1947 to (74.61, -29.48, -1.37) mm, rotated rx 180 ry 0 rz 90 deg; joints [73.573, -16.104, 78.523, 0, 27.581, 73.573]
  MoveL 1948 to (75.68, -28.4, -1.78) mm, rotated rx 180 ry 0 rz 90 deg; joints [73.616, -16.067, 78.452, 0, 27.615, 73.616]
  MoveL 1949 to (76.48, -27.11, -2.19) mm, rotated rx 180 ry 0 rz 90 deg; joints [73.664, -16.037, 78.406, 0, 27.631, 73.664]
  MoveL 1950 to (76.98, -25.68, -2.59) mm, rotated rx 180 ry 0 rz 90 deg; joints [73.712, -16.015, 78.386, 0, 27.629, 73.712]
  MoveL 1951 to (77.12, -24.17, -3) mm, rotated rx -180 ry 0 rz 90 deg; joints [73.76, -16.001, 78.395, 0, 27.607, 73.76]
  MoveL 1952 to (77.12, -5.21, -3) mm, rotated rx 180 ry 0 rz 90 deg; joints [74.347, -16.122, 78.806, 0, 27.317, 74.347]
  MoveL 1953 to (76.99, -2.37, -3) mm, rotated rx 180 ry 0 rz 90 deg; joints [74.434, -16.143, 78.876, 0, 27.267, 74.434]
  MoveL 1954 to (76.93, -1.88, -3) mm, rotated rx -180 ry 0 rz 90 deg; joints [74.448, -16.147, 78.89, 0, 27.257, 74.448]
  MoveC 1955 to (73.45, 2.01, -3) mm, rotated rx 180 ry 0 rz 90 deg; joints [74.54, -16.248, 79.236, 0, 27.012, 74.54] to (68.23, 2.31, -3) mm, rotated rx 180 ry 0 rz 90 deg; joints [74.504, -16.364, 79.635, 0, 26.729, 74.504]
  MoveC 1956 to (67.48, 1.76, -3) mm, rotated rx 180 ry 0 rz 90 deg; joints [74.48, -16.377, 79.68, 0, 26.697, 74.48] to (66.85, 1.08, -3) mm, rotated rx 180 ry 0 rz 90 deg; joints [74.453, -16.386, 79.713, 0, 26.673, 74.453]
  MoveL 1957 to (65.86, -0.21, -3) mm, rotated rx 180 ry 0 rz 90 deg; joints [74.404, -16.4, 79.76, 0, 26.64, 74.404]
  MoveL 1958 to (49.75, -22.31, -3) mm, rotated rx -180 ry 0 rz 90 deg; joints [73.569, -16.609, 80.488, 0, 26.12, 73.569]
  MoveC 1959 to (48.48, -26.09, -3) mm, rotated rx -180 ry 0 rz 90 deg; joints [73.438, -16.612, 80.499, 0, 26.113, 73.438] to (49.83, -29.85, -3) mm, rotated rx 180 ry 0 rz 90 deg; joints [73.334, -16.559, 80.316, 0, 26.244, 73.334]
  MoveL 1960 to (50.64, -30.8, -3) mm, rotated rx -180 ry 0 rz 90 deg; joints [73.312, -16.536, 80.235, 0, 26.301, 73.312]
  MoveL 1961 to (65.86, -48.01, -3) mm, rotated rx 180 ry 0 rz 90 deg; joints [72.921, -16.093, 78.707, 0, 27.387, 72.921]
  MoveL 1962 to (67.25, -49.5, -3) mm, rotated rx 180 ry 0 rz 90 deg; joints [72.889, -16.052, 78.568, 0, 27.485, 72.889]
  MoveC 1963 to (69.31, -50.78, -3) mm, rotated rx -180 ry 0 rz 90 deg; joints [72.869, -15.998, 78.382, 0, 27.615, 72.869] to (71.73, -50.82, -3) mm, rotated rx -180 ry 0 rz 90 deg; joints [72.89, -15.943, 78.198, 0, 27.745, 72.89]
  MoveL 1964 to (72.19, -50.7, -3) mm, rotated rx 180 ry 0 rz 90 deg; joints [72.899, -15.934, 78.166, 0, 27.768, 72.899]
  MoveC 1965 to (75.06, -49.14, -3) mm, rotated rx -180 ry 0 rz 90 deg; joints [72.973, -15.88, 77.985, 0, 27.895, 72.973] to (76.88, -46.45, -3) mm, rotated rx 180 ry 0 rz 90 deg; joints [73.073, -15.857, 77.909, 0, 27.948, 73.073]
  MoveC 1966 to (77.07, -44.79, -3) mm, rotated rx -180 ry 0 rz 90 deg; joints [73.125, -15.864, 77.933, 0, 27.932, 73.125] to (77.12, -43.12, -3) mm, rotated rx -180 ry 0 rz 90 deg; joints [73.177, -15.875, 77.967, 0, 27.907, 73.177]
  MoveL 1967 to (77.12, -24.17, -3) mm, rotated rx -180 ry 0 rz 90 deg; joints [73.76, -16.001, 78.395, 0, 27.607, 73.76]
  MoveL 1968 to (69.57, -24.17, -3) mm, rotated rx -180 ry 0 rz 90 deg; joints [73.692, -16.169, 78.966, 0, 27.203, 73.692]
  MoveL 1969 to (69.57, -24.17, 0) mm, rotated rx 180 ry 0 rz 90 deg; joints [73.692, -16.32, 79.068, 0, 27.252, 73.692]
  Establecer velocidad (1000.0 mm/s)
  MoveL 1970 to (69.57, -24.17, 10) mm, rotated rx -180 ry 0 rz 90 deg; joints [73.692, -16.82, 79.404, 0, 27.417, 73.692]
  Establecer velocidad (66.7 mm/s)
  MoveL 1971 to (37.53, 7.97, 10) mm, rotated rx 180 ry 0 rz 90 deg; joints [74.413, -17.697, 82.462, 0, 25.236, 74.413]
